(* CODESYS project CtaAppSensor_1.0.0.4.library
   Description: Sensor Library der CTA
   Version: 1.0.0.4
   Title: CtaAppSensor
   Author: SIS
   LanguageModelAttribute: qualified-access-only
   DocFormat: reStructuredText
   Placeholder: CtaAppSensor
   CompiledLibraryCompatibilityVersion: CODESYS V3.5 SP16 Patch 3
   Company: CTA
   DefaultNamespace: CtaAppSensor

Project tree, tasks and I/O mapping:
  libraries: Standard, 3.5.18.0 (System); CtaAppBmk, 1.0.0.0 (CTA); CtaAppReport, 1.0.0.2 (CTA); CtaSysConfig, 1.0.0.2 (CTA); CtaAppFilter, 1.0.0.0 (CTA); VisuSymbols, 4.5.0.0 (System); VisuDialogs, * (System); CtaSysSensorReCalculation, 1.0.0.0 (CTA); CtaVisSymbols, 1.0.0.0 (CTA); CtaAppInfluxLog, 1.0.0.1 (CTA); CtaSysIO, 1.0.0.1 (CTA); CtaVisHelp, 1.0.0.0 (CTA); CtaAppLeistungventile, 1.0.0.0 (CTA); CtaAppModbusSpezifikation, 1.0.0.0 (CTA)
  40 Visualizations/
    COLLECTOR/
      visualisation VIS_SENSOR_COLLECTOR
      visualisation VIS_SENSOR_COLLECTOR_TEMP
      Help Funktionen/
        visualisation SelSort
        visualisation SortPfeil
    ICON/
      SENSOR_FLAT/
        SENSOR_FLAT_TXT_RIGHT/
          ABOVE/
            visualisation VIS_SENSOR_FLAT_RigthAboveCheckIsEnabled
            visualisation VIS_SENSOR_FLAT_RIGHT_ABOVE
            visualisation VIS_SENSOR_FLAT_RigthAboveCheckQuerry
          BELOW/
            visualisation VIS_SENSOR_FLAT_RIGHT_BELOW
            visualisation VIS_SENSOR_FLAT_RigthBelowCheckIsEnabled
            visualisation VIS_SENSOR_FLAT_RigthBelowCheckQuerry
          MIDDLE/
            visualisation VIS_SENSOR_FLAT_RIGHT_MIDDLE
            visualisation VIS_SENSOR_FLAT_RigthMiddleCheckIsEnabled
            visualisation VIS_SENSOR_FLAT_RigthMiddleCheckQuerry
        SENSOR_FLAT_TXT_LEFT/
          BELOW/
            visualisation VIS_SENSOR_FLAT_LEFT_BELOW
            visualisation VIS_SENSOR_FLAT_LeftBelowCheckIsEnabled
            visualisation VIS_SENSOR_FLAT_LeftBelowCheckQuerry
          ABOVE/
            visualisation VIS_SENSOR_FLAT_LeftAboveCheckQuerry
            visualisation VIS_SENSOR_FLAT_LEFT_ABOVE
            visualisation VIS_SENSOR_FLAT_LeftAboveCheckIsEnabled
          MIDDLE/
            visualisation VIS_SENSOR_FLAT_LeftMiddleCheckIsEnabled
            visualisation VIS_SENSOR_FLAT_LeftMiddleCheckQuerry
            visualisation VIS_SENSOR_FLAT_LEFT_MIDDLE
      SENSOR_BASE/
        ICON/
          Round/
            visualisation SensorRound
          Flat/
            visualisation SensorFlat
          Value/
            visualisation ValueDwnUp
            visualisation ValueUpDwn
      SENSOR_ROUND/
        SENSOR_ROUND_TXT_RIGHT/
          ABOVE/
            visualisation VIS_SENSOR_ROUND_RIGHT_ABOVE
            visualisation VIS_SENSOR_ROUND_RightAboveCheckIsEnabled
            visualisation VIS_SENSOR_ROUND_RightAboveCheckQuerry
          BELOW/
            visualisation VIS_SENSOR_ROUND_RIGHT_BELOW
            visualisation VIS_SENSOR_ROUND_RightBelowCheckQuerry
            visualisation VIS_SENSOR_ROUND_RightBelowCheckIsEnabled
        SENSOR_ROUNF_TXT_LEFT/
          ABOVE/
            visualisation VIS_SENSOR_ROUND_LEFT_ABOVE
            visualisation VIS_SENSOR_ROUND_LeftAboveCheckIsEnabled
            visualisation VIS_SENSOR_ROUND_LeftAboveCheckQuerry
          BELOW/
            visualisation VIS_SENSOR_ROUND_LEFT_BELOW
            visualisation VIS_SENSOR_ROUND_LeftBelowCheckIsEnabled
            visualisation VIS_SENSOR_ROUND_LeftBelowCheckQuerry
    POPUP/
      visualisation POPUP_SENSOR
      PARAMETER/
        visualisation VIS_SENSOR_PARAMETER
        visualisation VIS_SENSOR_PARAMETER_LISTE
        SENSOR_ParameterBase/
          visualisation VIS_SENSOR_PARAMETER_BASE0
          visualisation VIS_SENSOR_PARAMETER_BASE
        SENSOR_ReportManagement/
          visualisation Sensor_LowAlarm_Param
          visualisation Sensor_HighAlarm_Param
          visualisation Sensor_HighWarning_Param
          visualisation VIS_SENSOR_PARAMETER_REPORTMNG
          visualisation VIS_SENSOR_PARAMETER_REPORTMNG_1
          visualisation Sensor_LowWarning_Param
        SENSOR_InfluxDb/
          visualisation VIS_SENSOR_PARAMETER_TRENDLOG
          visualisation VIS_SENSOR_PARAMETER_TRENDLOG0
        SENSOR_Filter/
          visualisation VIS_SENSOR_PARAMETER_FILTER
          visualisation VIS_SENSOR_PARAMETER_FILTER_1
        IO_Parameter/
          visualisation VIS_SENSOR_IO_PARAMETER
      visualisation VIS_SENSOR_LISTE
      MANUAL/
        visualisation VIS_SENSOR_MANUAL
      OVERVIEW/
        visualisation VIS_SENSOR_OVERVIEW
        visualisation VIS_SENSOR_OVERVIEW0
      REPORTS/
        visualisation VIS_SENSOR_REPORTS
      BUS/
        visualisation Sensor_BUS_CS
        visualisation Sensor_BUS
        visualisation Sensor_BUS_SW0_Detail
        visualisation Sensor_BUS_SW1_Detail
        visualisation Sensor_BUS_SW2_Detail
        visualisation Sensor_BUS_SW3_Detail
  30 Program Organization Units/
    Abstracte Bausteine/
      function block fbSensorTabellenInfo [ST]: proStateSymbol, proSoftwareValue, proRawValue, proEnSymbol, proPhysicalValue
    fb's/
      Sensor/
        function block fbSensor [ST]: proModulType, actReport, proITF_REPORTMANAGER, actErrorCondition, proLockDown, proAvailable, proAcknowlege, proAtIconNr, actTrendLog, proEn, proEnSymbol, metSetReal, metSetBool, proIsEnabled, proIsError, proStateSymbol, proCountedError, proCountedInfo, proCountedWarning, actState, proInvertierung, proxErrorConditionValue, proConfigError, actConfig, P_scAnalogAlarm_fbxEnableOverflowAl, P_scAnalogAlarm_fbxEnableUnderflowAl, P_scBase_fbxEnable, P_scVisu_fbusiDezimalPos, P_scAlCondition_fbxEnable, P_scAlCondition_fbtDelayTillCondition, P_scHighAlarm_fbiRetryTillLock, P_scHighAlarm_fbiTypeOfAcknolage, P_scHighAlarm_fbrHysterese, P_scHighAlarm_fbrValue, P_scHighAlarm_fbtDelayTillAlarm, P_scHighAlram_fbxDoesAlarm, P_scHighWarning_fbrValue, P_scHighWarning_fbtDelayTillWarning, P_scHighWarning_fbxDoesWarning, P_scInfluxDb_fbxEnable, P_scLoAlarm_fbiRetryTillLock, P_scLoAlarm_fbiTypeOfAcknolage, P_scLoAlarm_fbrHysterese, P_scLoAlarm_fbrValue, P_scLoAlarm_fbtDelayTillAlarm, P_scLoAlarm_fbxDoesAlarm, P_scLoWarning_fbrValue, P_scLoWarning_fbtDelayTillWarning, P_scLoWarning_fbxDoesWarning, P_scManual_fbrManualOnY, P_scManual_fbuiManualControl, P_scManual_fbuiManualState, P_scManual_fbxAllowManualOn, P_scAlarmReset_fbtDealyTillReset, P_scFilter_fbrValue, P_scFilter_fbxEnabled, proSensorITF, proRawValue, FB_INIT, proSoftwareValue, proIsWarning, proIsHandOnOrOff, proIsReady, proHandOff, proHandOn, proHandOnY, proAuto, proManualTrue, proManualFalse, proValueInputType, metSetITF, actDigital, actAnalog, proPhysicalValue, actReCalculate, ITF_RC, actMbState, proModbusTest, proModbusStateWord, proModbusControllWord, prorValue
      Collector/
        function block fbSensor_Collector [ST]: metRegistry, proMin, proMax, proaySensorTabelle, proMissedBuffer, proBufferError, proayAntrieb, metSortArray, metGetAntriebITF
    fc's/
      function fcGetBigerStringValue [ST]
      AlarmControll/
        function fcHighControl [ST]
        function fcLowControl [ST]
      Visu/
        function fcCheckQuerryAndIconReturn [ST]
  00000000-0000-0000-0000-000000000000|D:\CoDeSys\LibrariesV3\trunk\Intern\CAA\CAA Template\3.4.0.0 draft\Placeholder.xml
  00000000-0000-0000-0000-000000000000|D:\CoDeSys\LibrariesV3\trunk\Intern\CAA\CAA Template\3.2.0.3 draft\Prefix.pdf
  00000000-0000-0000-0000-000000000000|D:\CoDeSys\LibrariesV3\trunk\Intern\CAA\CAA Template\3.5.2.0 draft\Placeholder.xml
  20 Structs/
    13 Globale Variablen/
      global variables GVL_SENSOR
    data type scParameter
    LowWarning/
      data type scLoWarning
    BASE/
      data type scBase
    Alarme/
      data type scAnalogAlarm
      Zusatzbedingungen/
        data type scAlCondition
      AlarmReset/
        data type scAlarmReset
    HighWarning/
      data type scHighWarning
    InfluxDb/
      data type scInfluxDb
    Filter/
      data type scFilter
    HighAlarm/
      data type scHighAlarm
    LowAlarm/
      data type scLoAlarm
    Manual/
      data type scManual
    data type enInputType
    Visu/
      data type scVisu
  50 Images/
  10 Documenation/
    global variables VersionHistory
    global variables readMe
  21 Interface/
    interface ITF_SENSOR_COLLECTOR: proBufferError, metGetAntriebITF, proMissedBuffer, proMin, proMax, proaySensorTabelle, metSortArray
    interface ITF_SENSOR_TABELLE_INFO: proRawValue, proSoftwareValue, proEnSymbol, proStateSymbol, proPhysicalValue
    interface ITF_SENSOR: proConfigError, P_scBase_fbxEnable, P_scVisu_fbusiDezimalPos, P_scManual_fbxAllowManualOn, P_scManual_fbuiManualState, P_scManual_fbuiManualControl, P_scManual_fbrManualOnY, P_scFilter_fbxEnabled, P_scFilter_fbrValue, P_scLoWarning_fbxDoesWarning, P_scLoWarning_fbrValue, P_scLoWarning_fbtDelayTillWarning, P_scLoAlarm_fbxDoesAlarm, P_scLoAlarm_fbrValue, P_scLoAlarm_fbrHysterese, P_scLoAlarm_fbtDelayTillAlarm, P_scLoAlarm_fbiRetryTillLock, P_scLoAlarm_fbiTypeOfAcknolage, P_scHighWarning_fbxDoesWarning, P_scHighWarning_fbrValue, P_scHighWarning_fbtDelayTillWarning, P_scHighAlram_fbxDoesAlarm, P_scHighAlarm_fbrValue, P_scHighAlarm_fbrHysterese, P_scHighAlarm_fbtDelayTillAlarm, P_scHighAlarm_fbiRetryTillLock, P_scHighAlarm_fbiTypeOfAcknolage, P_scInfluxDb_fbxEnable, P_scAnalogAlarm_fbxEnableOverflowAl, P_scAnalogAlarm_fbxEnableUnderflowAl, P_scAlCondition_fbxEnable, P_scAlCondition_fbtDelayTillCondition, P_scAlarmReset_fbtDealyTillReset, proSensorITF, proCountedError, proCountedInfo, proITF_REPORTMANAGER, proCountedWarning, proIsHandOnOrOff, proHandOn, proIsError, proIsWarning, proEn, proIsEnabled, proHandOff, proHandOnY, proIsReady, proAuto, proManualFalse, proManualTrue, proValueInputType, proxErrorConditionValue, proInvertierung, prorValue, proLockDown, proAvailable, proAcknowlege, proAtIconNr, ITF_RC, proModbusStateWord, proModbusTest, proModbusControllWord
  11 Library Parameter/
    global variables Parameter
  12 Konstanten/
    global variables GlobalKonstant
  60 Textlisten/
    text list Info
    Types/
      text list WarnungsStatus
      text list ValueInputType
    Reports/
      text list Error
      text list Warnung
  text list GlobalTextList
  5ce3da45-db07-42e7-a21c-a00fff4ed8f6|C:\Users\sis\Downloads\dip-switch.svg
  5ce3da45-db07-42e7-a21c-a00fff4ed8f6|C:\Users\sis\Downloads\lightning-bolt-circle.svg
  5ce3da45-db07-42e7-a21c-a00fff4ed8f6|C:\Users\sis\Downloads\sine-wave.svg
  5ce3da45-db07-42e7-a21c-a00fff4ed8f6|C:\Users\sis\Downloads\eye.svg
  5ce3da45-db07-42e7-a21c-a00fff4ed8f6|C:\Users\sis\Downloads\lan.svg
*)

// 20 Structs/scParameter
{attribute 'pack_mode' := '1'} 
TYPE scParameter :
    STRUCT
        scBase              :   scBase;
		scManual			:	scManual;
		scFilter			:	scFilter;
		scLoWarning			:	scLoWarning;
		scLoAlarm			:	scLoAlarm;
		scHighWarning		:	scHighWarning;
		scHighAlarm			:	scHighAlarm;
		scInfluxDb			:	scInfluxDb;
		scAnalogAlarm		:	scAnalogAlarm;
		scAlCondition		:	scAlCondition;
		scAlarmReset		:	scAlarmReset;
		scVisu				:	scVisu;
    END_STRUCT
END_TYPE

// 20 Structs/HighWarning/scHighWarning
TYPE scHighWarning :
	STRUCT
		fbxDoesWarning			:	CtaSysConfig.fbBOOL;
		fbrValue				:	CtaSysConfig.fbREAL;
		fbtDelayTillWarning		:	CtaSysConfig.fbTIME;	
	END_STRUCT
END_TYPE

// 20 Structs/HighAlarm/scHighAlarm
TYPE scHighAlarm :
	STRUCT
		fbxDoesAlarm			:	CtaSysConfig.fbBOOL;
		fbrValue				:	CtaSysConfig.fbREAL;
		fbrHysterese			:	CtaSysConfig.fbREAL;
		fbtDeleayTillAlarm		:	CtaSysConfig.fbTIME;
		fbiRetryTillLock		:	CtaSysConfig.fbINT;
		fbiTypeOfAcknolage		:	CtaSysConfig.fbINT;
	END_STRUCT
END_TYPE

// 20 Structs/LowAlarm/scLoAlarm
TYPE scLoAlarm :
	STRUCT
		fbxDoesAlarm			:	CtaSysConfig.fbBOOL;
		fbrValue				:	CtaSysConfig.fbREAL;
		fbrHysterese			:	CtaSysConfig.fbREAL;
		fbtDeleayTillAlarm		:	CtaSysConfig.fbTIME;
		fbiRetryTillLock		:	CtaSysConfig.fbINT;
		fbiTypeOfAcknolage		:	CtaSysConfig.fbINT;
	END_STRUCT
END_TYPE

// 20 Structs/LowWarning/scLoWarning
TYPE scLoWarning :
	STRUCT
		fbxDoesWarning			:	CtaSysConfig.fbBOOL;
		fbrValue				:	CtaSysConfig.fbREAL;
		fbtDelayTillWarning		:	CtaSysConfig.fbTIME;		
	END_STRUCT
END_TYPE

// 20 Structs/Alarme/scAnalogAlarm
TYPE scAnalogAlarm :
	STRUCT
		fbxEnableOverflowAl		:	CtaSysConfig.fbBOOL;
		fbxEnableUnderflowAl	:	CtaSysConfig.fbBOOL;
	END_STRUCT
END_TYPE

// 20 Structs/Filter/scFilter
TYPE scFilter :
	STRUCT
		fbxEnabled	:	CtaSysConfig.fbBOOL;
		fbrValue	:	CtaSysConfig.fbREAL;
	END_STRUCT
END_TYPE

// 20 Structs/BASE/scBase
{attribute 'pack_mode' := '1'} 
TYPE scBase :
    STRUCT
        fbxEnable       :   CtaSysConfig.fbBOOL;
    END_STRUCT
END_TYPE

// 20 Structs/InfluxDb/scInfluxDb
{attribute 'pack_mode' := '1'} 
TYPE scInfluxDb :
    STRUCT
        fbxEnable       :   CtaSysConfig.fbBOOL;
    END_STRUCT
END_TYPE

// 20 Structs/Alarme/Zusatzbedingungen/scAlCondition
TYPE scAlCondition :
	STRUCT
		fbxEnable				:	CtaSysConfig.fbBOOL;
		fbtDelayTillCondition	:	CtaSysConfig.fbTIME;
	END_STRUCT
END_TYPE

// 20 Structs/Alarme/AlarmReset/scAlarmReset
TYPE scAlarmReset :
	STRUCT
		fbtDelayTillReset	:	CtaSysConfig.fbTIME;		
	END_STRUCT
END_TYPE

// 20 Structs/Manual/scManual
TYPE scManual :
	STRUCT
		fbxAlowManualOn		:	CtaSysConfig.fbBOOL;
		fbuiManualState		:	CtaSysConfig.fbUINT;
		fbuiManualControl	:	CtaSysConfig.fbUINT;
		fbrManualOnY		:	CtaSysConfig.fbREAL;
	END_STRUCT
END_TYPE

// 20 Structs/enInputType
{attribute 'qualified_only'}
{attribute 'strict'}
TYPE enInputType :
(
	Default := 0,
	AnalogInput,
	DigitalInput,
	Analog_ITF_Input,
	Digital_ITF_Input	
);
END_TYPE

// 20 Structs/Visu/scVisu
TYPE scVisu :
	STRUCT
		fbusiDezimalPos		:	CtaSysConfig.fbUSINT;
	END_STRUCT
END_TYPE

// 10 Documenation/VersionHistory
(* 

.. image:: ../../Images/CTA_Logo.jpg
   :align: right
   :width: 15% 

**Vorlage**   


============ =========== =========== ============================================
**Date**     **Version** **Author**  **Change**
------------ ----------- ----------- --------------------------------------------
04.03.2021   0.0.0.0     SIS         Vorlage erstellt

============ =========== =========== ============================================


*)
VAR_GLOBAL
    stInfo : STRING:= '0.0.0.0, Vorlage, CTA';
END_VAR

// 10 Documenation/readMe
(*

**ReadMe**
 
|	**Empfehlung**
|
|	Bibliothek CtaAppSensor zur auswertung von Sensoren
|	Instanzieren Sie den CtaAppSensor.fbSensor in ihrem Funktionsbaustein oder POU beispielsweise als fbTFühlX (X = Nr.) 
|	Deklarieren Sie die Struktur Variable welche als Parameter und zur ansteuerung dienen wie im Code beispiel.
|  
| *Beispiel* 

+-----------------------+---------------------------------------------------------------------------------------------------------------------------------------------------------------------------------------------------------------------------------------------------------------------------------------------------------------------------------------------------------------------------------------------------------------------------------------+
| Beschreibung          |  Code                                                                                                                                                                                                                                                                                                                                                                                                                                 |
+=======================+=======================================================================================================================================================================================================================================================================================================================================================================================================================================+
| POU oder SmFb         | .. code-block:: codesys                                                                                                                                                                                                                                                                                                                                                                                                               |
|                       |                                                                                                                                                                                                                                                                                                                                                                                                                                       |
|                       |	// Deklaration als VAR im POU oder dem selbsterstellten Funktionsbaustein                                                                                                                                                                                                                                                                                                                                                        	|
|                       |   VAR   																																																				 																																																				|
|						|	    (*Temperaturfühler 1*)																																																		 																																																	|
|						|		fbTFühl1			: CtaAppSensor.fbSensor;                                                                                                                                                                                                                                                                                                                                                               						|
|			 			|	END_VAR                                                                                                                                                                                                                                                                                                                                                                                                                          	|
+-----------------------+---------------------------------------------------------------------------------------------------------------------------------------------------------------------------------------------------------------------------------------------------------------------------------------------------------------------------------------------------------------------------------------------------------------------------------------+
| Code für Init         | .. code-block:: codesys                                                                                                                                                                                                                                                                                                                                                                                                               |
|                       |   																																																					 																																																				|
|			 			|	// Kopieren des nachfolgenden Codes in eine Action zur Initialisierung der Parameter. Zum Beispiel actConfig.																																																				 																										|
|                       |	{region "Parameter Temperaturfühler 1"}                                                                                                                                                                                                                                                                                                                                                                                             |
|			 			|		(*Basis*)                                                                                                                                                                                                                                                                                                                                                                                                                       |
|						|		fbTFühl1.scParameter.scBase.fbxEnable                			(_WertInit :=  TRUE																		 );		//P1 Ein- Ausschalten des Sensors                                                                                                                                                                                                                               |
|						|		(*Handansteuerung*)                                                                                                                                                                                                                                                                                                                                                                                                             |
|						|		fbTFühl1.scParameter.scManual.fbxAlowManualOn					(_WertInit := FALSE																		 );     //P2 Handansteuerung zulassen / nicht zulassen                                                                                                                                                                                                                  |
|						|		fbTFühl1.scParameter.scManual.fbuiManualState					(_WertInit :=	  0									, _MinInit :=     0, _MaxInit:=     2);     //P3 Ansteuerungsmodus des Sensors (auto, manuell, gesperrt)                                                                                                                                                                                                    |
|						|		fbTFühl1.scParameter.scManual.fbuiManualControl					(_WertInit :=     0									, _MinInit :=     0, _MaxInit:=     1);     //P4 Ansteuerungsignal des Sensors (TRUE,FALSE)                                                                                                                                                                                                                 |
|						|		fbTFühl1.scParameter.scManual.fbrManualOnY						(_WertInit :=   0.0									, _MinInit :=      , _MaxInit:=      );     //P5 Manueller Stellwert für den SEnsor                                                                                                                                                                                                                         |
|						|		(*Filter*)                                                                                                                                                                                                                                                                                                                                                                                                                      |
|						|		fbTFühl1.scParameter.scFilter.fbxEnabled						(_WertInit := FALSE																		 );		//P6 Ein- Ausschalten des Filters                                                                                                                                                                                                                               |
|						|		fbTFühl1.scParameter.scFilter.fbrValue							(_WertInit :=   0.0									, _MinInit :=      , _MaxInit:=      );		//P7 Filterwert                                                                                                                                                                                                                                                 |
|						|		(*LowWarning*)                                                                                                                                                                                                                                                                                                                                                                                                                  |
|						|		fbTFühl1.scParameter.scLoWarning.fbxDoesWarning					(_WertInit := FALSE																		 );		//P8 Ein- Ausschalten der LowWarning                                                                                                                                                                                                                            |
|						|		fbTFühl1.scParameter.scLoWarning.fbrValue						(_WertInit :=   0.0									, _minInit :=      , _maxInit:= 	 );		//P9 Wert bei welcher die LowWarning ausgelöst wird                                                                                                                                                                                                             |
|						|		fbTFühl1.scParameter.scLoWarning.fbtDelayTillWarning			(_WertInit :=  T#0S									, _minInit :=      , _maxInit:=      );		//P10 Verzögerungszeit für die Ausgabe des LowWarining Fehlers                                                                                                                                                                                                  |
|						|		(*LowAlarm*)                                                                                                                                                                                                                                                                                                                                                                                                                    |
|						|		fbTFühl1.scParameter.scLoAlarm.fbxDoesAlarm						(_WertInit := FALSE																		 );		//P11 Ein- Ausschalten des LowAlarm                                                                                                                                                                                                                             |
|						|		fbTFühl1.scParameter.scLoAlarm.fbrValue							(_WertInit :=   0.0									, _minInit :=      , _maxInit:= 	 );		//P12 Wert bei welchem der LowAlarm ausgelöst wird                                                                                                                                                                                                              |
|						|		fbTFühl1.scParameter.scLoAlarm.fbrHysterese						(_WertInit :=   0.0									, _minInit :=      , _maxInit:= 	 );		//P13 Histerese welche zur Rücksetung des Fehlers erreicht werden muss                                                                                                                                                                                          |
|						|		fbTFühl1.scParameter.scLoAlarm.fbtDeleayTillAlarm				(_WertInit :=  T#0S									, _minInit :=      , _maxInit:= 	 );		//P14 Verzögerungszeit für die Ausgabe des LowAlarm Fehlers                                                                                                                                                                                                     |
|						|		fbTFühl1.scParameter.scLoAlarm.fbiTypeOfAcknolage				(_WertInit :=     0 								, _minInit :=     0, _maxInit:=     2);		//P15 Art der Quittierung des Fehlers (auto, quittierned, quittiernd bis n Meldung)                                                                                                                                                                             |
|						|		fbTFühl1.scParameter.scLoAlarm.fbiRetryTillLock					(_WertInit :=     3									, _minInit :=     0, _maxInit:=     5);		//P16 Maximale Anzahl Wiederholungen bis zu Sperrung der Anlage                                                                                                                                                                                                 |
|						|		(*HighWarning*)                                                                                                                                                                                                                                                                                                                                                                                                                 |
|						|		fbTFühl1.scParameter.scHighWarning.fbxDoesWarning				(_WertInit := FALSE																		 );		//P17 Ein- Ausschalten der HighWarning                                                                                                                                                                                                                    		|
|						|		fbTFühl1.scParameter.scHighWarning.fbrValue						(_WertInit :=   0.0									, _minInit :=      , _maxInit:= 	 );		//P18 Wert bei welcher die HighWarning ausgelöst wird                                                                                                                                                                                                     		|
|						|		fbTFühl1.scParameter.scHighWarning.fbtDelayTillWarning			(_WertInit :=  T#0S									, _minInit := 	   , _maxInit:= 	 );		//P19 Verzögerungszeit für die Ausgabe des HighWarining Fehlers                                                                                                                                                                                           		|
|						|		(*HighAlarm*)                                                                                                                                                                                                                                                                                                                                                                                                                   |
|						|		fbTFühl1.scParameter.scHighAlarm.fbxDoesAlarm					(_WertInit := FALSE															 			 );		//P20 Ein- Ausschalten des HighAlarm                                                                                                                                                                                                                            |
|						|		fbTFühl1.scParameter.scHighAlarm.fbrValue						(_WertInit :=   0.0									, _minInit :=      , _maxInit:=      );		//P21 Wert bei welchem der HighAlarm ausgelöst wird                                                                                                                                                                                                             |
|						|		fbTFühl1.scParameter.scHighAlarm.fbrHysterese					(_WertInit :=   0.0									, _minInit :=      , _maxInit:= 	 );		//P22 Histerese welche zur Rücksetung des Fehlers erreicht werden muss                                                                                                                                                                                          |
|						|		fbTFühl1.scParameter.scHighAlarm.fbtDeleayTillAlarm				(_WertInit :=  T#0S									, _minInit :=      , _maxInit:=      );		//P23 Verzögerungszeit für die Ausgabe des HighAlarm Fehlers                                                                                                                                                                                                    |
|						|		fbTFühl1.scParameter.scHighAlarm.fbiTypeOfAcknolage				(_WertInit := 	  0 								, _minInit :=      , _maxInit:=     2);		//P24 Art der Quittierung des Fehlers (auto, quittierned, quittiernd bis n Meldung)                                                                                                                                                                             |
|						|		fbTFühl1.scParameter.scHighAlarm.fbiRetryTillLock				(_WertInit :=     3									, _minInit :=      , _maxInit:=     5);		//P25 Maximale Anzahl Wiederholungen bis zu Sperrung der Anlage                                                                                                                                                                                                 |
|						|		(*Überlauf, Unterlauf*)                                                                                                                                                                                                                                                                                                                                                                                                         |
|						|		fbTFühl1.scParameter.scAnalogAlarm.fbxEnableOverflowAl			(_WertInit :=  TRUE																		 );		//P26 Ein- Ausschalten des Überlauf- Alarms                                                                                                                                                                                                                     |
|						|		fbTFühl1.scParameter.scAnalogAlarm.fbxEnableUnderflowAl			(_WertInit :=  TRUE																		 );		//P27 Ein- Ausschalten des Unterlauf- Alrams                                                                                                                                                                                                                    |
|						|		(*Zusatzbedingung*)                                                                                                                                                                                                                                                                                                                                                                                                             |
|						|		fbTFühl1.scParameter.scAlCondition.fbxEnable 					(_WertInit := FALSE																		 );		//P28 Ein- Ausschalten der Zusatzbedingung                                                                                                                                                                                                                      |
|						|		fbTFühl1.scParameter.scAlCondition.fbtDelayTillCondition		(_WertInit :=  T#0S									, _minInit :=      ,_maxInit:=       );		//P29 Verzögerung für die Zusatzbedingung                                                                                                                                                                                                                       |
|						|		(*Alarmrücksetzung*)                                                                                                                                                                                                                                                                                                                                                                                                            |
|						|		fbTFühl1.scParameter.scAlarmReset.fbtDelayTillReset				(_WertInit := T#24H									, _minInit :=      ,_maxInit:=       );		//P30 Verzögerung für die Fehlerrücksetzung                                                                                                                                                                                                                     |
|						|		(*Trendlog*)                                                                                                                                                                                                                                                                                                                                                                                                                    |
|						|		fbTFühl1.scParameter.scInfluxDb.fbxEnable            			(_WertInit := TRUE																		 );		//P31 Aktiverung / Deaktivierung der Trenddaten														 																																							|
|						|		(*Visu*)                                                                                                                                                                                                                                                                                                                                                                                                                    	|
|						|		fbTFühl1.scParameter.scVisu.fbusiDezimalPos            			(_WertInit :=     1									, _minInit := 0     , _maxInit:=    3);		//P32 Dezimalstellen auf Visu													 																																												|
|						|	{endregion}                                                                                                                                                      																																																																    | 
|						|																																																																																																										|
+-----------------------+---------------------------------------------------------------------------------------------------------------------------------------------------------------------------------------------------------------------------------------------------------------------------------------------------------------------------------------------------------------------------------------------------------------------------------------+
*)                                                                                                                                                                                                                                                                                                                                                                                                                                                               
VAR_GLOBAL
	xReadMeDone              :   BOOL; 
END_VAR

// 20 Structs/13 Globale Variablen/GVL_SENSOR
{attribute 'qualified_only'}
VAR_GLOBAL
    fbSENSOR_COLLECTOR	:   fbSensor_Collector;   
    xValidData          :   BOOL;
END_VAR

// 11 Library Parameter/Parameter
{attribute 'qualified_only'}
VAR_GLOBAL CONSTANT
    iMaxSensor :   INT   := 60;         // Maximale Anzahl verwendeter AT-Bausteine    
END_VAR

// 12 Konstanten/GlobalKonstant
{attribute 'qualified_only'}
VAR_GLOBAL CONSTANT 	
	stReportTextListError   : CtaAppReport.stReportTextList := 'CtaAppSensor.Error';
	stReportTextListWarning : CtaAppReport.stReportTextList := 'CtaAppSensor.Warnung';
	stReportTextListInfo    : CtaAppReport.stReportTextList := 'CtaAppSensor.Info';	
END_VAR

// 30 Program Organization Units/fb's/Sensor/fbSensor
FUNCTION_BLOCK fbSensor EXTENDS fbSensorTabellenInfo IMPLEMENTS ITF_SENSOR 
VAR_INPUT
    xAlCondition               	:   BOOL;
	xEnHandMode					:	BOOL;
 	rSimValue					:	REAL;
END_VAR                         
VAR_OUTPUT 
    xValue                      :   BOOL;
    rValue						:   REAL;
	rValueRC					:	REAL;
	xIsHandMode					:	BOOL;
END_VAR                 
VAR 
	(*Inputs*)
	ITF_IO_IN					:	CtaSysIO.ITF_IO;
	xValueIn					:	BOOL;
	rValueIn					:	REAL;	
	(* Input Type*)
	xIsITF						:	BOOL;
	xIsBool						:	BOOL;
	xIsReal						:	BOOL;
    stAlternateUnit				:	STRING(5);                
    (* State Intern*)
	xIsDigital					:	BOOL;
	_ITF_DI						: 	CtaSysIO.ITF_DI;
	_ITF_AI						:	CtaSysIO.ITF_AI; 	
	rValueTemp					:	REAL;
	xValueTemp					:	BOOL;
	enValueInputType			:   enInputType;     
    scEWI                       :   CtaAppReport.scReportNr; 
	xIsEnabled					:	BOOL;                
	xConfigError                :   BOOL;
	uiIconNr					:	UINT;
	xOk							:	BOOL;
	(* Modbus *)
    xModbusTest                 :   BOOL;
    ayMbControllWord            :   ARRAY[0..3] OF WORD;
    ayMbStateWord               :   ARRAY[0..3] OF WORD;	
    (* Parameter *)
    fbConfigFile                :   CtaSysConfig.fbConfigFile;
    scParameter                 :   scParameter;	
    (* Reports *)		
    fbReportManager			    :   CtaAppReport.fbReportManager;      
    difor					    :	DINT;                                                                    
    ayErrorReporter				:	ARRAY[1..7] OF CtaAppReport.fbReporter;
	ayWarningReporter			:	ARRAY[1..6] OF CtaAppReport.fbReporter; 	
	_xIsWarning					:	BOOL;
	xIsWarning					:	BOOL;	
	_xIsError					:	BOOL;
	xIsError					:	BOOL;		
	xLoWarning					:	BOOL;
	xLoAlarm					:	BOOL;
	xHiWarning					:	BOOL;
	xHiAlarm					:	BOOL;	
	(* Trendlogs *)
	fbTrendxValue				:	CtaAppInfluxLog.FB_LOG_NODE_BOOL;
	fbTrendrValue				:	CtaAppInfluxLog.FB_LOG_NODE_REAL;
	fbTrendrVaueUnfiltered		:	CtaAppInfluxLog.FB_LOG_NODE_REAL;
	fbTrendrVaueRC				:	CtaAppInfluxLog.FB_LOG_NODE_REAL;
	(* Filter *)
	fbFilter					:	CtaAppFilter.fbImpulsFilter;	
	rValueUngefiltert			:	REAL;	
    (* Collector *)
    diArrayPosition             :   DINT;
	xManualValue				:	BOOL;
	xIsHandOff					:	BOOL;
	xIsHandOn					:	BOOL;
	xIsAuto						:	BOOL;
	xIsHand						:	BOOL;
	TON_DelayAlCondition		: 	TON;
	xErrorConditionOn			: 	BOOL;
	
	xErrorConditionAttached		:	BOOL;
	(*Calculator *)				
	ITF_RC_QUERY				:	CtaSysSensorReCalculation.ITF_SENSOR_RE_CALCULATE;
END_VAR

(* Config *)
actConfig();

(* Sensor Command *)
IF xIsEnabled AND NOT xConfigError THEN
	IF xIsITF THEN
		IF __QUERYINTERFACE(ITF_IO_IN,_ITF_DI) THEN
			enValueInputType := enInputType.Digital_ITF_Input;
			actDigital();
		ELSIF __QUERYINTERFACE(ITF_IO_IN,_ITF_AI) THEN
			enValueInputType := enInputType.Analog_ITF_Input;
			actAnalog();
		END_IF
		
	ELSIF xIsBool THEN
		enValueInputType := enInputType.DigitalInput;
		actDigital();
	ELSIF xIsReal THEN
		enValueInputType := enInputType.AnalogInput;
		actAnalog();
	ELSE
		enValueInputType := enInputType.Default;		
	END_IF	
	
	(* Al Condition *)
    actErrorCondition();	
    (* EWI *)
    actReport();    

	(* Recalculation *)
	actReCalculate();             
ELSE
    IF xConfigError THEN
        (* EWI *)
      actReport();         
	END_IF;
END_IF;

(* State *)
actState();
actMbState();
(* InfluxDB *)
actTrendLog();

PROPERTY proModulType : CtaSysIO.enModuleType
GET
proModulType := ITF_IO_IN.proModuleType;
END_GET
END_PROPERTY

ACTION actReport:
(* EWI Manager *)
fbReportManager(	stErrorInitReportTextListIn		:=	ADR(GlobalKonstant.stReportTextListError),
					stWarningInitReportTextListIn	:=	ADR(GlobalKonstant.stReportTextListWarning),
					stInfoInitReportTextListIn		:=	ADR(GlobalKonstant.stReportTextListInfo),
					scReportNr						:=	scEWI);

IF xIsBool OR (xIsITF AND __QUERYINTERFACE (ITF_IO_IN,_ITF_DI))  THEN
	(* Errors *)                        
        (* Alarm Minimalwert erreicht *)
        ayErrorReporter[1].proPrio  := 2;
        ayErrorReporter[1].metReport(     		xSetReportIn					:= xErrorConditionOn AND scParameter.scLoAlarm.fbxDoesAlarm.proValue AND xLoAlarm,
												iReportID						:= 1,
												enReportTypeIn					:= CtaAppReport.enReportType.Error,  
												enReportAcknowledgeTypeIn   	:= scParameter.scLoAlarm.fbiTypeOfAcknolage.proValue,
												tDelay							:= scParameter.scLoAlarm.fbtDeleayTillAlarm.proValue, 
												ITF_BMK_IN						:= THIS^,			              
												pstReportTextListIn				:= ADR(GlobalKonstant.stReportTextListError),
												stOptionalReportText		    := '',   
												iRetryTilReportLock 		    := scParameter.scLoAlarm.fbiRetryTillLock.proValue, 
												xResetCount         		    := FALSE,  
												tReset						    := scParameter.scAlarmReset.fbtDelayTillReset.proValue); 		

        (* Alarm Maximalwert erreicht *)    
        ayErrorReporter[2].proPrio  := 2;
        ayErrorReporter[2].metReport(     		xSetReportIn					:= xErrorConditionOn AND scParameter.scHighAlarm.fbxDoesAlarm.proValue AND xHiAlarm,
												iReportID						:= 2,
												enReportTypeIn					:= CtaAppReport.enReportType.Error,  
												enReportAcknowledgeTypeIn   	:= scParameter.scHighAlarm.fbiTypeOfAcknolage.proValue,
												tDelay							:= scParameter.scHighAlarm.fbtDeleayTillAlarm.proValue, 
												ITF_BMK_IN						:= THIS^,			              
												pstReportTextListIn				:= ADR(GlobalKonstant.stReportTextListError),
												stOptionalReportText		    := '',   
												iRetryTilReportLock 		    := scParameter.scHighAlarm.fbiRetryTillLock.proValue,
												xResetCount         		    := FALSE, 
	                               				tReset						    := scParameter.scAlarmReset.fbtDelayTillReset.proValue); 		

(* Warnungen *)      
        (* Warnung Minimalwert erreicht *)      
        ayWarningReporter[1].proPrio := 2;
        ayWarningReporter[1].metReport(			xSetReportIn					:= xErrorConditionOn AND scParameter.scLoWarning.fbxDoesWarning.proValue AND xLoWarning,
												iReportID						:= 1,
												enReportTypeIn					:= CtaAppReport.enReportType.Warning,  
												enReportAcknowledgeTypeIn   	:= CtaAppReport.enReportAcknowledgeType.Auto,
												tDelay							:= scParameter.scLoWarning.fbtDelayTillWarning.proValue, 
												ITF_BMK_IN						:= THIS^,			              
												pstReportTextListIn				:= ADR(GlobalKonstant.stReportTextListWarning),
												stOptionalReportText		    := '',   
												iRetryTilReportLock 		    := 0, 
												xResetCount         		    := FALSE,  
												tReset						    := T#0S);                       
                                  
        (* Warnung Maxiwalwert erreicht *)
        ayWarningReporter[2].proPrio := 2;
        ayWarningReporter[2].metReport(			xSetReportIn					:= xErrorConditionOn AND scParameter.scHighWarning.fbxDoesWarning.proValue AND xHiWarning,
												iReportID						:= 2,
												enReportTypeIn					:= CtaAppReport.enReportType.Warning,  
												enReportAcknowledgeTypeIn   	:= CtaAppReport.enReportAcknowledgeType.Auto,
												tDelay							:= scParameter.scHighWarning.fbtDelayTillWarning.proValue, 
												ITF_BMK_IN						:= THIS^,			              
												pstReportTextListIn				:= ADR(GlobalKonstant.stReportTextListWarning),
												stOptionalReportText		    := '',   
												iRetryTilReportLock 		    := 0, 
												xResetCount         		    := FALSE,
												tReset						    := T#0S);  
		
ELSIF xIsReal OR (xIsITF AND __QUERYINTERFACE (ITF_IO_IN,_ITF_AI)) THEN
(* Errors *)                        
	(* Alarm Minimalwert erreicht *)
	ayErrorReporter[3].proPrio  := 2;
	ayErrorReporter[3].metReport(     		xSetReportIn					:= xErrorConditionOn AND scParameter.scLoAlarm.fbxDoesAlarm.proValue AND xLoAlarm,
											iReportID						:= 3,
											enReportTypeIn					:= CtaAppReport.enReportType.Error,  
											enReportAcknowledgeTypeIn   	:= scParameter.scLoAlarm.fbiTypeOfAcknolage.proValue,
											tDelay							:= scParameter.scLoAlarm.fbtDeleayTillAlarm.proValue, 
											ITF_BMK_IN						:= THIS^,			              
											pstReportTextListIn				:= ADR(GlobalKonstant.stReportTextListError),
											stOptionalReportText		    := '',   
											iRetryTilReportLock 		    := scParameter.scLoAlarm.fbiRetryTillLock.proValue, 
											xResetCount         		    := FALSE,  
											tReset						    := scParameter.scAlarmReset.fbtDelayTillReset.proValue); 		

	(* Alarm Maximalwert erreicht *)    
	ayErrorReporter[4].proPrio  := 2;
	ayErrorReporter[4].metReport(     		xSetReportIn					:= xErrorConditionOn AND scParameter.scHighAlarm.fbxDoesAlarm.proValue AND xHiAlarm,
											iReportID						:= 4,
											enReportTypeIn					:= CtaAppReport.enReportType.Error,  
											enReportAcknowledgeTypeIn   	:= scParameter.scHighAlarm.fbiTypeOfAcknolage.proValue,
											tDelay							:= scParameter.scHighAlarm.fbtDeleayTillAlarm.proValue, 
											ITF_BMK_IN						:= THIS^,			              
											pstReportTextListIn				:= ADR(GlobalKonstant.stReportTextListError),
											stOptionalReportText		    := '',   
											iRetryTilReportLock 		    := scParameter.scHighAlarm.fbiRetryTillLock.proValue,
											xResetCount         		    := FALSE, 
											tReset						    := scParameter.scAlarmReset.fbtDelayTillReset.proValue); 
		
		(* Additional errors over interface*)
		IF NOT xIsReal THEN									
			(* Alarm Unterlauf *)
			ayErrorReporter[5].proPrio  := 2;
			ayErrorReporter[5].metReport(     		xSetReportIn					:= scParameter.scAnalogAlarm.fbxEnableUnderflowAl.proValue AND _ITF_AI.proAlUnterlauf,
													iReportID						:= 5,
													enReportTypeIn					:= CtaAppReport.enReportType.Error,  
													enReportAcknowledgeTypeIn   	:= CtaAppReport.enReportAcknowledgeType.Auto,
													tDelay							:= T#0S, 
													ITF_BMK_IN						:= THIS^,			              
													pstReportTextListIn				:= ADR(GlobalKonstant.stReportTextListError),
													stOptionalReportText		    := '',   
													iRetryTilReportLock 		    := 0, 
													xResetCount         		    := FALSE,  
													tReset						    := T#0S); 		
		
			(* Alarm Überlauf *)    
			ayErrorReporter[6].proPrio  := 2;
			ayErrorReporter[6].metReport(     		xSetReportIn					:= scParameter.scAnalogAlarm.fbxEnableOverflowAl.proValue AND _ITF_AI.proAlUeberlauf,
													iReportID						:= 6,
													enReportTypeIn					:= CtaAppReport.enReportType.Error,  
													enReportAcknowledgeTypeIn   	:= CtaAppReport.enReportAcknowledgeType.Auto,
													tDelay							:= T#0S, 
													ITF_BMK_IN						:= THIS^,			              
													pstReportTextListIn				:= ADR(GlobalKonstant.stReportTextListError),
													stOptionalReportText		    := '',   
													iRetryTilReportLock 		    := 0,
													xResetCount         		    := FALSE, 
													tReset						    := T#0S);
		END_IF
			
(* Warnungen *)      
	(* Warnung Minimalwert erreicht *)      
	ayWarningReporter[3].proPrio := 2;
	ayWarningReporter[3].metReport(			xSetReportIn					:= xErrorConditionOn AND scParameter.scLoWarning.fbxDoesWarning.proValue AND xLoWarning,
											iReportID						:= 3,
											enReportTypeIn					:= CtaAppReport.enReportType.Warning,  
											enReportAcknowledgeTypeIn   	:= CtaAppReport.enReportAcknowledgeType.Auto,
											tDelay							:= scParameter.scLoWarning.fbtDelayTillWarning.proValue, 
											ITF_BMK_IN						:= THIS^,			              
											pstReportTextListIn				:= ADR(GlobalKonstant.stReportTextListWarning),
											stOptionalReportText		    := '',   
											iRetryTilReportLock 		    := 0, 
											xResetCount         		    := FALSE,  
											tReset						    := T#0S);                       
							  
	(* Warnung Maxiwalwert erreicht *)
	ayWarningReporter[4].proPrio := 2;
	ayWarningReporter[4].metReport(			xSetReportIn					:= xErrorConditionOn AND scParameter.scHighWarning.fbxDoesWarning.proValue AND xHiWarning,
											iReportID						:= 4,
											enReportTypeIn					:= CtaAppReport.enReportType.Warning,  
											enReportAcknowledgeTypeIn   	:= CtaAppReport.enReportAcknowledgeType.Auto,
											tDelay							:= scParameter.scHighWarning.fbtDelayTillWarning.proValue, 
											ITF_BMK_IN						:= THIS^,			              
											pstReportTextListIn				:= ADR(GlobalKonstant.stReportTextListWarning),
											stOptionalReportText		    := '',   
											iRetryTilReportLock 		    := 0, 
											xResetCount         		    := FALSE,
											tReset						    := T#0S);
END_IF

(* Config Error *)    
ayErrorReporter[7].proPrio  := 1;
ayErrorReporter[7].metReport(     		xSetReportIn					:= xConfigError,
										iReportID						:= 7,
										enReportTypeIn					:= CtaAppReport.enReportType.Error,  
										enReportAcknowledgeTypeIn   	:= CtaAppReport.enReportacknowledgeType.Quit,
										tDelay							:= T#1S, 
										ITF_BMK_IN						:= THIS^,			              
										pstReportTextListIn				:= ADR(GlobalKonstant.stReportTextListError),
										stOptionalReportText		    := '',   
										iRetryTilReportLock 		    := 0, 
										xResetCount         		    := FALSE,  
										tReset						    := T#24H);                            

		
(* Warnung Hand Aus *)      
ayWarningReporter[5].proPrio := 3;  
ayWarningReporter[5].proHandLokal :=    xIsHandOff; 
ayWarningReporter[5].metReport(			xSetReportIn					:= xIsHandOff,
										iReportID						:= 5,
										enReportTypeIn					:= CtaAppReport.enReportType.Warning,  
										enReportAcknowledgeTypeIn   	:= CtaAppReport.enReportAcknowledgeType.Auto,
										tDelay							:= T#0S, 
										ITF_BMK_IN						:= THIS^,			              
										pstReportTextListIn				:= ADR(GlobalKonstant.stReportTextListWarning),
										stOptionalReportText		    := '',   
										iRetryTilReportLock 		    := 0, 
										xResetCount         		    := FALSE,  
										tReset						    := T#24H);                                  
                                
(* Warnung Hand Ein *)    
ayWarningReporter[6].proPrio := 3; 
ayWarningReporter[6].proHandLokal :=    xIsHandOn;
ayWarningReporter[6].metReport(			xSetReportIn					:= xIsHandOn OR xIsHandMode,
										iReportID						:= 6,
										enReportTypeIn					:= CtaAppReport.enReportType.Warning,  
										enReportAcknowledgeTypeIn   	:= CtaAppReport.enReportAcknowledgeType.Auto,
										tDelay							:= T#0S, 
										ITF_BMK_IN						:= THIS^,			              
										pstReportTextListIn				:= ADR(GlobalKonstant.stReportTextListWarning),
										stOptionalReportText		    := '',   
										iRetryTilReportLock 		    := 0, 
										xResetCount         		    := FALSE,  
										tReset						    := T#24H);                                           
	
(* Sync Reports *)                                         
FOR difor := LOWER_BOUND(ayErrorReporter,1) TO UPPER_BOUND(ayErrorReporter,1) DO
	fbReportManager.metSyncReporter(ayErrorReporter[difor]);	
END_FOR;
FOR difor := LOWER_BOUND(ayWarningReporter,1) TO UPPER_BOUND(ayWarningReporter,1) DO
	fbReportManager.metSyncReporter(ayWarningReporter[difor]);	
END_FOR;
                                                                          
_xIsError   := scEWI.iError <> 0;
_xIsWarning := scEWI.iWarning <> 0;
END_ACTION

PROPERTY proITF_REPORTMANAGER : CtaAppReport.ITF_REPORTMANAGER
GET
proITF_REPORTMANAGER := fbReportManager;
END_GET
END_PROPERTY

ACTION actErrorCondition:
//  Zeitverzögerung bis die Alarmierung Freigegeben wird


IF scParameter.scAlCondition.fbxEnable.proValue			THEN
	TON_DelayAlCondition(   PT:=    scParameter.scAlCondition.fbtDelayTillCondition.proValue,
							IN:=	xAlCondition,
							Q=>     xErrorConditionOn);  
             
ELSE
xErrorConditionOn		:=TRUE;	
END_IF
END_ACTION

{attribute 'monitoring' := 'variable'}
PROPERTY proLockDown : BOOL
GET
proLockDown := proIsError;
END_GET
END_PROPERTY

{attribute 'monitoring' := 'variable'}
PROPERTY proAvailable : BOOL
GET
proAvailable := proIsReady;
END_GET
END_PROPERTY

{attribute 'monitoring' := 'variable'}
PROPERTY proAcknowlege : BOOL
GET
proAcknowlege := xValue AND NOT proIsError ;
END_GET
END_PROPERTY

PROPERTY proAtIconNr : UINT
SET
uiIconNr := proAtIconNr;
END_SET
GET
proAtIconNr:= uiIconNr;
END_GET
END_PROPERTY

ACTION actTrendLog:
(* Istwert bool *)
fbTrendxValue.ENABLE		:= 	scParameter.scBase.fbxEnable.proValue AND 
								scParameter.scInfluxDb.fbxEnable.proValue;
fbTrendxValue.KEY           :=  CONCAT(stObjID,'_xValue');
fbTrendxValue.SET_VALUE     :=  xValue;

(* Istwert real *)
fbTrendrValue.ENABLE		:=	scParameter.scBase.fbxEnable.proValue AND 
								scParameter.scInfluxDb.fbxEnable.proValue;
fbTrendrValue.KEY           :=  CONCAT(stObjID,'_rValue');
fbTrendrValue.SET_VALUE     :=  rValue;

IF (xIsITF AND  __QUERYINTERFACE (ITF_IO_IN,_ITF_AI)) OR xIsReal THEN
	(* Istwert real ungefiltert*)
	fbTrendrVaueUnfiltered.ENABLE		:=	scParameter.scBase.fbxEnable.proValue AND 
											scParameter.scInfluxDb.fbxEnable.proValue;
	fbTrendrVaueUnfiltered.KEY			:=  CONCAT(stObjID,'_rValueUnfiltered');
	fbTrendrVaueUnfiltered.SET_VALUE	:= 	rValueUngefiltert;
ELSE
	(* Istwert real ungefiltert*)
	fbTrendrVaueUnfiltered.ENABLE		:=	FALSE;
	fbTrendrVaueUnfiltered.KEY			:=  CONCAT(stObjID,'_rValueUnfiltered');
	fbTrendrVaueUnfiltered.SET_VALUE	:= 	rValueUngefiltert;	
END_IF;

IF __QUERYINTERFACE(ITF_RC_QUERY,ITF_RC_QUERY) THEN
	(* Recalculatet Value Enable*)
	fbTrendrVaueRC.ENABLE				:=	scParameter.scBase.fbxEnable.proValue AND 
											scParameter.scInfluxDb.fbxEnable.proValue;
	fbTrendrVaueRC.KEY					:=  CONCAT(stObjID,'_rValueRecalculatet');
	fbTrendrVaueRC.SET_VALUE			:= 	rValueRC;
ELSE
	(* Recalculatet Value Disable*)
	fbTrendrVaueRC.ENABLE				:=	FALSE;
	fbTrendrVaueRC.KEY					:=  CONCAT(stObjID,'_rValueRecalculatet');
	fbTrendrVaueRC.SET_VALUE			:= 	rValueRC;	
END_IF;
END_ACTION

PROPERTY proEn : BOOL
SET
xIsEnabled := proEn;
END_SET
GET
proEn := xIsEnabled;
END_GET
END_PROPERTY

PROPERTY proEnSymbol : STRING
GET
IF xIsEnabled THEN
    proEnSymbol := 'CtaVisSymbols.ImagePool.CheckboxChecked_blue';
ELSE    
    proEnSymbol := 'CtaVisSymbols.ImagePool.CheckboxUnchecked_withe'; 
END_IF;
END_GET
END_PROPERTY

METHOD metSetReal
VAR_INPUT
	rRealIn				:	REAL;
	stAlternateUnitIn	:	STRING(5);
END_VAR
rValueIn 		:= rRealIn;
xIsITF 			:= FALSE;
xIsBool 		:= FALSE;
xIsReal 		:= TRUE;
stAlternateUnit := stAlternateUnitIn;
END_METHOD

METHOD metSetBool
VAR_INPUT
	xBoolIn		:  BOOL;
END_VAR
xValueIn := xBoolIn;
xIsITF	:= FALSE;
xIsBool := TRUE;
xIsReal := FALSE;
END_METHOD

PROPERTY proIsEnabled : BOOL
GET
proIsEnabled := xIsEnabled;
END_GET
END_PROPERTY

PROPERTY proIsError : BOOL
GET
proIsError := xIsError;
END_GET
END_PROPERTY

PROPERTY proStateSymbol : STRING
GET
IF xIsError THEN
    proStateSymbol := 'CtaVisSymbols.ImagePool.CtaError';
ELSE    
    IF xIsWarning THEN
        IF scEWI.iWarning = 5 THEN
            proStateSymbol := 'CtaVisSymbols.ImagePool.front_hand_Yellow_Off';
        ELSIF scEWI.iWarning = 6 THEN
            proStateSymbol := 'CtaVisSymbols.ImagePool.front_hand_Yellow';
        ELSE
            proStateSymbol := 'CtaVisSymbols.ImagePool.CtaWarning';
        END_IF;
     ELSE
         proStateSymbol := '';
	 END_IF
END_IF;
END_GET
END_PROPERTY

PROPERTY proCountedError : INT
GET
proCountedError := fbReportManager.proAnzError;
END_GET
END_PROPERTY

PROPERTY proCountedInfo : INT
GET
proCountedInfo := fbReportManager.proAnzInfo;
END_GET
END_PROPERTY

PROPERTY proCountedWarning : INT
GET
proCountedWarning := fbReportManager.proAnzWarning;
END_GET
END_PROPERTY

ACTION actState:
xIsWarning      := _xIsWarning;         
xIsError        := _xIsError;        
xIsEnabled      := scParameter.scBase.fbxEnable.proValue;         
xIsHandOn       := scParameter.scManual.fbuiManualState.proValue = 2;         
xIsHandOff      := scParameter.scManual.fbuiManualState.proValue = 1;          
xIsAuto         := scParameter.scManual.fbuiManualState.proValue = 0;
xManualValue	:= scParameter.scManual.fbuiManualControl.proValue = 1 AND scParameter.scManual.fbuiManualControl.proValue <> 0;
xIsHand        	:= xIsHandOn OR xEnHandMode OR xIsHandOff;
END_ACTION

PROPERTY proInvertierung : BOOL;
GET
IF __QUERYINTERFACE(_ITF_DI,_ITF_DI) THEN	
	proInvertierung := 	TO_BOOL(CtaSysConfig.fcGetEnumerationId(_ITF_DI.P_scfbDI_fbxInvert));
ELSE
	proInvertierung := FALSE;
END_IF
END_GET
END_PROPERTY

PROPERTY proxErrorConditionValue : BOOL
GET
proxErrorConditionValue := xErrorConditionOn;
END_GET
END_PROPERTY

PROPERTY proConfigError : BOOL
GET
proConfigError := xConfigError;
END_GET
END_PROPERTY

ACTION actConfig:
(* Config Fb *)
fbConfigFile();

(* Base Parameter *)
scParameter.scBase.fbxEnable                			(_usiParaNr :=  1, ItfConfigFb := fbConfigFile);

(* Manual *)
scParameter.scManual.fbxAlowManualOn					(_usiParaNr :=  2, itfConfigFb := fbConfigFile);
scParameter.scManual.fbuiManualState					(_usiParaNr :=  3, itfConfigFb := fbConfigFile);
scParameter.scManual.fbuiManualControl					(_usiParaNr :=  4, itfConfigFb := fbConfigFile);
scParameter.scManual.fbrManualOnY						(_usiParaNr :=  5, itfConfigFb := fbConfigFile);

(* Filter *)
scParameter.scFilter.fbxEnabled							(_usiParaNr :=  6, itfConfigFb := fbConfigFile);
scParameter.scFilter.fbrValue							(_usiParaNr :=  7, itfConfigFb := fbConfigFile);

(* Low warning *)
scParameter.scLoWarning.fbxDoesWarning					(_usiParaNr :=  8, itfConfigFb := fbConfigFile);
scParameter.scLoWarning.fbrValue						(_usiParaNr :=  9, itfConfigFb := fbConfigFile);
scParameter.scLoWarning.fbtDelayTillWarning				(_usiParaNr := 10, itfConfigFb := fbConfigFile);

(* Low alarm *)
scParameter.scLoAlarm.fbxDoesAlarm						(_usiParaNr := 11, itfConfigFb := fbConfigFile);
scParameter.scLoAlarm.fbrValue							(_usiParaNr := 12, itfConfigFb := fbConfigFile);
scParameter.scLoAlarm.fbrHysterese						(_usiParaNr := 13, itfConfigFb := fbConfigFile);
scParameter.scLoAlarm.fbtDeleayTillAlarm				(_usiParaNr := 14, itfConfigFb := fbConfigFile);
scParameter.scLoAlarm.fbiTypeOfAcknolage				(_usiParaNr := 15, itfConfigFb := fbConfigFile, _MinInit := 0 , _MaxInit := 2);
scParameter.scLoAlarm.fbiRetryTillLock					(_usiParaNr := 16, itfConfigFb := fbConfigFile);

(* High warning *)
scParameter.scHighWarning.fbxDoesWarning				(_usiParaNr := 17, itfConfigFb := fbConfigFile);
scParameter.scHighWarning.fbrValue						(_usiParaNr := 18, itfConfigFb := fbConfigFile);
scParameter.scHighWarning.fbtDelayTillWarning			(_usiParaNr := 19, itfConfigFb := fbConfigFile);

(* High alarm *)
scParameter.scHighAlarm.fbxDoesAlarm					(_usiParaNr := 20, itfConfigFb := fbConfigFile);
scParameter.scHighAlarm.fbrValue						(_usiParaNr := 21, itfConfigFb := fbConfigFile);
scParameter.scHighAlarm.fbrHysterese					(_usiParaNr := 22, itfConfigFb := fbConfigFile);
scParameter.scHighAlarm.fbtDeleayTillAlarm				(_usiParaNr := 23, itfConfigFb := fbConfigFile);
scParameter.scHighAlarm.fbiTypeOfAcknolage				(_usiParaNr := 24, itfConfigFb := fbConfigFile, _MinInit := 0 , _MaxInit := 2);
scParameter.scHighAlarm.fbiRetryTillLock				(_usiParaNr := 25, itfConfigFb := fbConfigFile);

(* Alarm *)
scParameter.scAnalogAlarm.fbxEnableOverflowAl			(_usiParaNr := 26, itfConfigFb := fbConfigFile);
scParameter.scAnalogAlarm.fbxEnableUnderflowAl			(_usiParaNr := 27, itfConfigFb := fbConfigFile);

(* Alarm extra conditions *)
scParameter.scAlCondition.fbxEnable 					(_usiParaNr := 28, itfConfigFb := fbConfigFile);
scParameter.scAlCondition.fbtDelayTillCondition			(_usiParaNr := 29, itfConfigFb := fbConfigFile);

(* Alarm reset after... *)
scParameter.scAlarmReset.fbtDelayTillReset				(_usiParaNr := 30, itfConfigFb := fbConfigFile);

(* InfluxDb *)
scParameter.scInfluxDb.fbxEnable            			(_usiParaNr := 31, ItfConfigFb := fbconfigFile);

(* Visu *)
scParameter.scVisu.fbusiDezimalPos						(_usiParaNr := 32, ItfConfigFb := fbconfigFile, _minInit := 0, _maxInit := 3);

xConfigError := fbConfigFile.xError;
END_ACTION

PROPERTY P_scAnalogAlarm_fbxEnableOverflowAl : CtaSysConfig.ITF_DATATYPE
GET
P_scAnalogAlarm_fbxEnableOverflowAl:= scParameter.scAnalogAlarm.fbxEnableOverflowAl;
END_GET
END_PROPERTY

PROPERTY P_scAnalogAlarm_fbxEnableUnderflowAl : CtaSysConfig.ITF_DATATYPE
GET
P_scAnalogAlarm_fbxEnableUnderflowAl := scParameter.scAnalogAlarm.fbxEnableUnderflowAl;
END_GET
END_PROPERTY

PROPERTY P_scBase_fbxEnable : CtaSysConfig.ITF_DATATYPE
GET
P_scBase_fbxEnable := scParameter.scBase.fbxEnable;
END_GET
END_PROPERTY

PROPERTY P_scVisu_fbusiDezimalPos : CtaSysConfig.ITF_DATATYPE
GET
P_scVisu_fbusiDezimalPos := scParameter.scVisu.fbusiDezimalPos;
END_GET
END_PROPERTY

PROPERTY P_scAlCondition_fbxEnable : CtaSysConfig.ITF_DATATYPE
GET
P_scAlCondition_fbxEnable := scParameter.scAlCondition.fbxEnable;
END_GET
END_PROPERTY

PROPERTY P_scAlCondition_fbtDelayTillCondition : CtaSysConfig.ITF_DATATYPE
GET
P_scAlCondition_fbtDelayTillCondition := scParameter.scAlCondition.fbtDelayTillCondition;
END_GET
END_PROPERTY

PROPERTY P_scHighAlarm_fbiRetryTillLock : CtaSysConfig.ITF_DATATYPE
GET
P_scHighAlarm_fbiRetryTillLock := scParameter.scHighAlarm.fbiRetryTillLock;
END_GET
END_PROPERTY

PROPERTY P_scHighAlarm_fbiTypeOfAcknolage : CtaSysConfig.ITF_DATATYPE
GET
P_scHighAlarm_fbiTypeOfAcknolage := scParameter.scHighAlarm.fbiTypeOfAcknolage;
END_GET
END_PROPERTY

PROPERTY P_scHighAlarm_fbrHysterese : CtaSysConfig.ITF_DATATYPE
GET
P_scHighAlarm_fbrHysterese := scParameter.scHighAlarm.fbrHysterese;
END_GET
END_PROPERTY

PROPERTY P_scHighAlarm_fbrValue : CtaSysConfig.ITF_DATATYPE
GET
P_scHighAlarm_fbrValue := scParameter.scHighAlarm.fbrValue;
END_GET
END_PROPERTY

PROPERTY P_scHighAlarm_fbtDelayTillAlarm : CtaSysConfig.ITF_DATATYPE
GET
P_scHighAlarm_fbtDelayTillAlarm := scParameter.scHighAlarm.fbtDeleayTillAlarm;
END_GET
END_PROPERTY

PROPERTY P_scHighAlram_fbxDoesAlarm : CtaSysConfig.ITF_DATATYPE
GET
P_scHighAlram_fbxDoesAlarm := scParameter.scHighAlarm.fbxDoesAlarm;
END_GET
END_PROPERTY

PROPERTY P_scHighWarning_fbrValue : CtaSysConfig.ITF_DATATYPE
GET
P_scHighWarning_fbrValue := scParameter.scHighWarning.fbrValue;
END_GET
END_PROPERTY

PROPERTY P_scHighWarning_fbtDelayTillWarning : CtaSysConfig.ITF_DATATYPE
GET
P_scHighWarning_fbtDelayTillWarning := scParameter.scHighWarning.fbtDelayTillWarning;
END_GET
END_PROPERTY

PROPERTY P_scHighWarning_fbxDoesWarning : CtaSysConfig.ITF_DATATYPE
GET
P_scHighWarning_fbxDoesWarning := scParameter.scHighWarning.fbxDoesWarning;
END_GET
END_PROPERTY

PROPERTY P_scInfluxDb_fbxEnable : CtaSysConfig.ITF_DATATYPE
GET
P_scInfluxDb_fbxEnable := scParameter.scInfluxDb.fbxEnable;
END_GET
END_PROPERTY

PROPERTY P_scLoAlarm_fbiRetryTillLock : CtaSysConfig.ITF_DATATYPE
GET
P_scLoAlarm_fbiRetryTillLock := scParameter.scLoAlarm.fbiRetryTillLock;
END_GET
END_PROPERTY

PROPERTY P_scLoAlarm_fbiTypeOfAcknolage : CtaSysConfig.ITF_DATATYPE
GET
P_scLoAlarm_fbiTypeOfAcknolage := scParameter.scLoAlarm.fbiTypeOfAcknolage;
END_GET
END_PROPERTY

PROPERTY P_scLoAlarm_fbrHysterese : CtaSysConfig.ITF_DATATYPE
GET
P_scLoAlarm_fbrHysterese := scParameter.scLoAlarm.fbrHysterese;
END_GET
END_PROPERTY

PROPERTY P_scLoAlarm_fbrValue : CtaSysConfig.ITF_DATATYPE
GET
P_scLoAlarm_fbrValue := scParameter.scLoAlarm.fbrValue;
END_GET
END_PROPERTY

PROPERTY P_scLoAlarm_fbtDelayTillAlarm : CtaSysConfig.ITF_DATATYPE
GET
P_scLoAlarm_fbtDelayTillAlarm := scParameter.scLoAlarm.fbtDeleayTillAlarm;
END_GET
END_PROPERTY

PROPERTY P_scLoAlarm_fbxDoesAlarm : CtaSysConfig.ITF_DATATYPE
GET
P_scLoAlarm_fbxDoesAlarm := scParameter.scLoAlarm.fbxDoesAlarm;
END_GET
END_PROPERTY

PROPERTY P_scLoWarning_fbrValue : CtaSysConfig.ITF_DATATYPE
GET
P_scLoWarning_fbrValue := scParameter.scLoWarning.fbrValue;
END_GET
END_PROPERTY

PROPERTY P_scLoWarning_fbtDelayTillWarning : CtaSysConfig.ITF_DATATYPE
GET
P_scLoWarning_fbtDelayTillWarning := scParameter.scLoWarning.fbtDelayTillWarning;
END_GET
END_PROPERTY

PROPERTY P_scLoWarning_fbxDoesWarning : CtaSysConfig.ITF_DATATYPE
GET
P_scLoWarning_fbxDoesWarning := scParameter.scLoWarning.fbxDoesWarning;
END_GET
END_PROPERTY

PROPERTY P_scManual_fbrManualOnY : CtaSysConfig.ITF_DATATYPE
GET
P_scManual_fbrManualOnY := scParameter.scManual.fbrManualOnY;
END_GET
END_PROPERTY

PROPERTY P_scManual_fbuiManualControl : CtaSysConfig.ITF_DATATYPE
GET
P_scManual_fbuiManualControl := scParameter.scManual.fbuiManualControl;
END_GET
END_PROPERTY

PROPERTY P_scManual_fbuiManualState : CtaSysConfig.ITF_DATATYPE
GET
P_scManual_fbuiManualState := scParameter.scManual.fbuiManualState;
END_GET
END_PROPERTY

PROPERTY P_scManual_fbxAllowManualOn : CtaSysConfig.ITF_DATATYPE
GET
P_scManual_fbxAllowManualOn := scParameter.scManual.fbxAlowManualOn;
END_GET
END_PROPERTY

PROPERTY P_scAlarmReset_fbtDealyTillReset : CtaSysConfig.ITF_DATATYPE
GET
P_scAlarmReset_fbtDealyTillReset := scParameter.scAlarmReset.fbtDelayTillReset;
END_GET
END_PROPERTY

PROPERTY P_scFilter_fbrValue : CtaSysConfig.ITF_DATATYPE
GET
P_scFilter_fbrValue := scParameter.scFilter.fbrValue;
END_GET
END_PROPERTY

PROPERTY P_scFilter_fbxEnabled : CtaSysConfig.ITF_DATATYPE
GET
P_scFilter_fbxEnabled := scParameter.scFilter.fbxEnabled;
END_GET
END_PROPERTY

PROPERTY proSensorITF : CtaSysIO.ITF_IO;
GET
proSensorITF := ITF_IO_IN;
END_GET
END_PROPERTY

PROPERTY proRawValue : STRING
GET
IF xIsITF THEN
	IF __QUERYINTERFACE (_ITF_DI,_ITF_DI) THEN	
		proRawValue := TO_STRING(_ITF_DI.proValue);
	ELSIF __QUERYINTERFACE(_ITF_AI,_ITF_AI) THEN
		IF _ITF_AI.proModuleType = CtaSysIO.enModuleType.DC_0_10V_IN THEN
			proRawValue :=	CONCAT(TO_STRING(_ITF_AI.proPhysicalValue),' v');
		ELSIF _ITF_AI.proModuleType = CtaSysIO.enModuleType.DC_4_20mA_IN THEN
			proRawValue :=	CONCAT(TO_STRING(_ITF_AI.proPhysicalValue),' mA');
		ELSIF _ITF_AI.proModuleType = CtaSysIO.enModuleType.ohm THEN
			proRawValue :=	CONCAT(TO_STRING(_ITF_AI.proPhysicalValue),' °C');
		ELSE
			proRawValue := '';	
		END_IF
	ELSE
		proRawValue := '';			
	END_IF	
ELSIF xIsBool THEN
	proRawValue := TO_STRING(xValueIn);
ELSIF xIsReal THEN
	proRawValue := TO_STRING(rValueIn);
ELSE
	proRawValue := '';	
END_IF
END_GET
END_PROPERTY

//FB_Init ist immer implizit verfügbar und wird primär für die Initialisierung verwendet.
//Der Rückgabewert wird nicht ausgewertet. Für gezielte Einflussnahme können Sie
//die Methoden explizit deklarieren und darin mit dem Standard-Initialisierungscode 
//zusätzlichen Code bereitstellen. Sie können den Rückgabewert auswerten.
METHOD FB_INIT: BOOL
VAR_INPUT    
bInitRetains: BOOL; // TRUE: Die Retain-Variablen werden initialisiert (Reset warm / Reset kalt)    
bInCopyCode: BOOL;  // TRUE: Die Instanz wird danach in den Kopiercode kopiert (Online-Change)
END_VAR
VAR
    ITF_SENSOR_THIS             :   ITF_SENSOR;
    ITF_SENSOR_QUERRY           :   ITF_SENSOR;
END_VAR
IF NOT bInCopyCode THEN
    ITF_SENSOR_THIS := THIS^;
    IF __QUERYINTERFACE(ITF_SENSOR_THIS,ITF_SENSOR_QUERRY) THEN
        diArrayPosition := GVL_SENSOR.fbSensor_Collector.metRegistry(ITF_SENSOR_QUERRY);
    END_IF;
END_IF;
END_METHOD

PROPERTY proSoftwareValue : STRING
GET
IF xIsBool OR ( xIsITF AND __QUERYINTERFACE (_ITF_DI,_ITF_DI)) THEN
	proSoftwareValue := TO_STRING(xValue);
ELSIF xIsReal THEN
	proSoftwareValue := CONCAT(TO_STRING(CTASYsCONFIG.fcRealToString(rValue,scparameter.scVisu.fbusiDezimalPos.usiValue)),stAlternateUnit);	 
ELSIF xIsITF AND __QUERYINTERFACE(_ITF_AI,_ITF_AI) THEN
	IF _ITF_AI.proModuleType = CtaSysIO.enModuleType.OHM THEN
		proSoftwareValue := CONCAT(TO_STRING(CTASYsCONFIG.fcRealToString(rValue,scparameter.scVisu.fbusiDezimalPos.usiValue)),'°C') ;
	ELSE
		proSoftwareValue := CONCAT(TO_STRING(CTASYsCONFIG.fcRealToString(rValue,scparameter.scVisu.fbusiDezimalPos.usiValue)),CtaSysConfig.fcGetValueFromDataType(_ITF_AI.P_scfbAI_fbstPhysicalUnit)) ;
	END_IF	
ELSE
	proSoftwareValue := '';
END_IF
END_GET
END_PROPERTY

PROPERTY proIsWarning : BOOL
GET
proIsWarning := xIsWarning;
END_GET
END_PROPERTY

PROPERTY proIsHandOnOrOff : BOOL
GET
proIsHandOnOrOff := xIsHand;
END_GET
END_PROPERTY

PROPERTY proIsReady : BOOL
GET
proIsReady := xIsEnabled AND NOT xIsError;
END_GET
END_PROPERTY

PROPERTY proHandOff : BOOL
SET
IF proHandOff THEN
	scParameter.scManual.fbuiManualState.proValue := 1;
END_IF
END_SET
GET
proHandOff := xIsHandOff;
END_GET
END_PROPERTY

PROPERTY proHandOn : BOOL
GET
proHandOn := xIsHandOn OR xIsHandMode;
END_GET
SET
IF proHandOn THEN
	scParameter.scManual.fbuiManualState.proValue := 2;
END_IF
END_SET
END_PROPERTY

PROPERTY proHandOnY : REAL
SET
scParameter.scManual.fbrManualOnY.proValue := proHandOnY;
END_SET
GET
proHandOnY := scParameter.scManual.fbrManualOnY.proValue;
END_GET
END_PROPERTY

PROPERTY proAuto : BOOL
SET
IF proAuto THEN
	scParameter.scManual.fbuiManualState.provalue := 0;
END_IF
END_SET
GET
proAuto := xIsAuto;
END_GET
END_PROPERTY

PROPERTY proManualTrue : BOOL
SET
IF proManualTrue THEN
	scParameter.scManual.fbuiManualControl.proValue := 1;
END_IF
END_SET
GET
proManualTrue := xManualValue;
END_GET
END_PROPERTY

PROPERTY proManualFalse : BOOL
SET
IF proManualFalse THEN
	scParameter.scManual.fbuiManualControl.proValue := 0;
END_IF
END_SET
GET
proManualFalse := NOT xManualValue;
END_GET
END_PROPERTY

PROPERTY proValueInputType : enInputType
GET
proValueInputType := enValueInputType;
END_GET
END_PROPERTY

METHOD metSetITF
VAR_INPUT
	ITF_IN		:	CtaSysIO.ITF_IO;
END_VAR
ITF_IO_IN := ITF_IN;
xIsITF 	:= TRUE;
xIsBool := FALSE;
xIsReal := FALSE;
END_METHOD

ACTION actDigital:
IF _ITF_DI <> 0 THEN
	xValueTemp := _ITF_DI.proValue;
ELSE
	xValueTemp := xValueIn;	
END_IF

(* Low Controll *)
xLoWarning      := fcLowControl(xEn   := scParameter.scLoWarning.fbxDoesWarning.proValue,
								rIst  := TO_REAL(xValueTemp),
								rLow  := 0,
								rHyst := 0,
								xTrig := 0);
								
xLoAlarm      	:= fcLowControl(xEn   := scParameter.scLoAlarm.fbxDoesAlarm.proValue,
								rIst  := TO_REAL(xValueTemp),
								rLow  := 0,
								rHyst := 0,
								xTrig := 0);

(* High Controll *)
xHiWarning     := fcHighControl(xEn   := scParameter.scHighWarning.fbxDoesWarning.proValue,
								rIst  := TO_REAL(xValueTemp),
								rHigh := 1,
								rHyst := 0,
								xTrig := 0);
								
xHiAlarm       := fcHighControl(xEn   := scParameter.scHighAlarm.fbxDoesAlarm.proValue,
								rIst  := TO_REAL(xValueTemp),
								rHigh := 1,
								rHyst := 0,
								xTrig := 0);

(* Hand Off *)
IF scParameter.scManual.fbuiManualState.proValue = 1 THEN
	xValue := NOT xValueTemp;	
	xIsHandMode := FALSE;
(* Hand On *)	
ELSIF scParameter.scManual.fbuiManualState.proValue <> 2 AND NOT xEnHandMode THEN
	(* Value *)
	xValue := xValueTemp;
	xIsHandMode := FALSE;
ELSE
	xValue := SEL(xEnHandMode,xManualValue,TO_BOOL(rSimValue));
	xIsHandMode := TRUE;
	
	IF NOT scParameter.scManual.fbxAlowManualOn.proValue AND NOT xEnHandMode THEN
		xValue := xValueTemp;
		xIsHandMode := FALSE;
	END_IF
END_IF

rValue := TO_REAL(xValue);
END_ACTION

ACTION actAnalog:
IF _ITF_AI <> 0 THEN	
	rValueUngefiltert      := _ITF_AI.proValue;
	xOk					   := _ITF_AI.proOK; 
ELSE	
	rValueUngefiltert      := rValueIn; 
END_IF
        
(* Low Controll *)
xLoWarning	:= fcLowControl(xEn   := scParameter.scLoWarning.fbxDoesWarning.proValue,
							rIst  := rValueUngefiltert,
							rLow  := scParameter.scLoWarning.fbrValue.proValue,
							rHyst := 0,
							xTrig := 0);
(* ToLow Controll *)
xLoAlarm    := fcLowControl(xEn   := scParameter.scLoAlarm.fbxDoesAlarm.proValue,
							rIst  := rValueUngefiltert,
							rlow  := scParameter.scLoAlarm.fbrValue.proValue,
							rHyst := scParameter.scLoAlarm.fbrHysterese.proValue,
							xTrig := xLoAlarm);
							
(* High Controll *)
xHiWarning := fcHighControl(xEn   := scParameter.scHighWarning.fbxDoesWarning.proValue,
							rIst  := rValueUngefiltert,
							rHigh := scParameter.scHighWarning.fbrValue.proValue,
							rHyst := 0,
							xTrig := 0);
(* ToHigh Controll *)
xHiAlarm   := fcHighControl(xEn   := scParameter.scHighAlarm.fbxDoesAlarm.proValue,
							rIst  := rValueUngefiltert,
							rHigh := scParameter.scHighAlarm.fbrValue.proValue,
							rHyst := scParameter.scHighAlarm.fbrHysterese.proValue,
							xTrig := xHiAlarm);
							
(* Filter *)
IF scParameter.scFilter.fbxEnabled.proValue THEN
	fbFilter   				   (rIn  	:= rValueUngefiltert,
								rFilter := scParameter.scFilter.fbrValue.proValue);
	(* Value Out*)
	rValueTemp  := fbFilter.rOut;
ELSE
	(* Value Out*)
	rValueTemp  := rValueUngefiltert;
END_IF

IF scParameter.scManual.fbuiManualState.proValue = 1 THEN
	rValue := 0;
	xIsHandMode := FALSE;
ELSIF scParameter.scManual.fbuiManualState.proValue <> 2 AND NOT xEnHandMode THEN
	rValue := rValueTemp;
	xIsHandMode := FALSE;
ELSE
	rValue := SEL(xEnHandMode,scParameter.scManual.fbrManualOnY.proValue,rSimValue);
	xIsHandMode := TRUE;
	
	IF NOT scParameter.scManual.fbxAlowManualOn.proValue AND NOT xEnHandMode THEN
		rValue := rValueTemp;
		xIsHandMode := FALSE;
	END_IF
END_IF

xValue  := scEWI.iError = 0 AND SEL(_ITF_AI <> 0,TRUE ,xOk);
END_ACTION

PROPERTY proPhysicalValue : STRING
GET
IF xIsITF THEN
	IF __QUERYINTERFACE (_ITF_AI,_ITF_AI)THEN
		proPhysicalValue := CONCAT(TO_STRING(_ITF_AI.proValue),CtaSysConfig.fcGetValueFromDataType(_ITF_AI.P_scfbAI_fbstPhysicalUnit));
	ELSIF __QUERYINTERFACE (_ITF_DI,_ITF_DI) THEN
		proPhysicalValue := TO_STRING(_ITF_DI.proValue);
	ELSE
		proPhysicalValue := '';
	END_IF
ELSIF xIsBool THEN
	proPhysicalValue := TO_STRING(xValueIn);
ELSIF xIsReal THEN
	proPhysicalValue :=TO_STRING(rValueIn);
ELSE
	proPhysicalValue := '';
END_IF
END_GET
END_PROPERTY

ACTION actReCalculate:
IF __QUERYINTERFACE(ITF_RC_QUERY,ITF_RC_QUERY) THEN
	ITF_RC_QUERY.VALUE := rValue;
	rValueRC := ITF_RC_QUERY.CALCULATET_VALUE;
ELSE
	rValueRC := rValue;
END_IF;
END_ACTION

PROPERTY ITF_RC : CtaSysSensorReCalculation.ITF_SENSOR_RE_CALCULATE
SET
ITF_RC_QUERY := ITF_RC;
END_SET
GET
ITF_RC := ITF_RC_QUERY;
END_GET
END_PROPERTY

ACTION actMbState:
IF NOT xModbusTest THEN
    (* State Word 0 Digital Info*)
    ayMbStateWord[0].00     := xValue;
    ayMbStateWord[0].01     := FALSE;
    ayMbStateWord[0].02     := FALSE;
    ayMbStateWord[0].03     := FALSE;
    ayMbStateWord[0].04     := FALSE;
    ayMbStateWord[0].05     := FALSE;
    ayMbStateWord[0].06     := FALSE;
    ayMbStateWord[0].07     := FALSE;
    ayMbStateWord[0].08     := xIsHand;
    ayMbStateWord[0].09     := xIsAuto;
    ayMbStateWord[0].10     := FALSE;
    ayMbStateWord[0].11     := FALSE;
    ayMbStateWord[0].12     := FALSE;
    ayMbStateWord[0].13     := FALSE;
    ayMbStateWord[0].14     := xIsWarning;
    ayMbStateWord[0].15     := xIsError;
	
	IF (enValueInputType = enInputType.DigitalInput) OR (enValueInputType = enInputType.Digital_ITF_Input) THEN
		(* State Word 1 setpoint*)
		ayMbStateWord[1]   	:= TO_WORD(TO_INT(xValue));
		(* State Word 2 actual value*)
		ayMbStateWord[3]	:= TO_WORD(TO_INT(xValue));
	ELSE
		 (* State Word 1 setpoint*)
		ayMbStateWord[1]   	:= TO_WORD(TO_INT(rValue * 10));
		(* State Word 2 actual value*)
		ayMbStateWord[2]	:= TO_WORD(TO_INT(rValueRC * 10));
		(* State Word 3 actual value*)
		ayMbStateWord[3]	:=	SEL(enValueInputType = enInputType.Analog_ITF_Input,TO_WORD(TO_INT(rValue * 10)),TO_WORD(TO_INT(_ITF_AI.proPhysicalValue * 10)));	
	END_IF
END_IF;
END_ACTION

PROPERTY proModbusTest : BOOL
SET
xModbusTest := proModbusTest;
END_SET
GET
proModbusTest := xModbusTest;
END_GET
END_PROPERTY

{warning disable C0410}
PROPERTY proModbusStateWord : REFERENCE TO ARRAY[0..3] OF WORD
{warning restore C0410}
GET
proModbusStateWord REF= ayMbStateWord;
END_GET
END_PROPERTY

{warning disable C0410}
PROPERTY proModbusControllWord : REFERENCE TO ARRAY[0..3] OF WORD
{warning restore C0410}
GET
proModbusControllWord REF= ayMbControllWord;
END_GET
END_PROPERTY

PROPERTY prorValue : REAL
GET
prorValue := rValue;
END_GET
END_PROPERTY

END_FUNCTION_BLOCK

// 30 Program Organization Units/Abstracte Bausteine/fbSensorTabellenInfo
{attribute 'hide'} 
FUNCTION_BLOCK INTERNAL ABSTRACT fbSensorTabellenInfo EXTENDS CtaAppBmk.fbBMK IMPLEMENTS ITF_SENSOR_TABELLE_INFO

PROPERTY proStateSymbol : STRING
GET
END_GET
END_PROPERTY

PROPERTY proSoftwareValue : STRING
GET
END_GET
END_PROPERTY

PROPERTY proRawValue : STRING
GET
END_GET
END_PROPERTY

PROPERTY proEnSymbol : STRING
GET
END_GET
END_PROPERTY

PROPERTY proPhysicalValue : STRING
GET
END_GET
END_PROPERTY

END_FUNCTION_BLOCK

// 21 Interface/ITF_SENSOR_TABELLE_INFO
INTERFACE INTERNAL ITF_SENSOR_TABELLE_INFO EXTENDS CtaAppBmk.ITF_BMK

PROPERTY proRawValue : STRING
GET
END_GET
END_PROPERTY

PROPERTY proSoftwareValue : STRING
GET
END_GET
END_PROPERTY

{attribute 'hide'} 
PROPERTY INTERNAL proEnSymbol : STRING
GET
END_GET
END_PROPERTY

{attribute 'hide'} 
PROPERTY INTERNAL proStateSymbol : STRING
GET
END_GET
END_PROPERTY

PROPERTY proPhysicalValue : STRING
GET
END_GET
END_PROPERTY

END_INTERFACE

// 21 Interface/ITF_SENSOR
INTERFACE ITF_SENSOR EXTENDS ITF_SENSOR_TABELLE_INFO , CtaAppModbusSpezifikation.ITF_MODBUS_SPEZIFIKATION

{attribute 'hide'} 
PROPERTY proConfigError : BOOL
GET
END_GET
END_PROPERTY

PROPERTY P_scBase_fbxEnable : CtaSysConfig.ITF_DATATYPE
GET
END_GET
END_PROPERTY

PROPERTY P_scVisu_fbusiDezimalPos : CtaSysConfig.ITF_DATATYPE
GET
END_GET
END_PROPERTY

PROPERTY P_scManual_fbxAllowManualOn : CtaSysConfig.ITF_DATATYPE
GET
END_GET
END_PROPERTY

PROPERTY P_scManual_fbuiManualState : CtaSysConfig.ITF_DATATYPE
GET
END_GET
END_PROPERTY

PROPERTY P_scManual_fbuiManualControl : CtaSysConfig.ITF_DATATYPE
GET
END_GET
END_PROPERTY

PROPERTY P_scManual_fbrManualOnY : CtaSysConfig.ITF_DATATYPE
GET
END_GET
END_PROPERTY

PROPERTY P_scFilter_fbxEnabled : CtaSysConfig.ITF_DATATYPE
GET
END_GET
END_PROPERTY

PROPERTY P_scFilter_fbrValue : CtaSysConfig.ITF_DATATYPE
GET
END_GET
END_PROPERTY

PROPERTY P_scLoWarning_fbxDoesWarning : CtaSysConfig.ITF_DATATYPE
GET
END_GET
END_PROPERTY

PROPERTY P_scLoWarning_fbrValue : CtaSysConfig.ITF_DATATYPE
GET
END_GET
END_PROPERTY

PROPERTY P_scLoWarning_fbtDelayTillWarning : CtaSysConfig.ITF_DATATYPE
GET
END_GET
END_PROPERTY

PROPERTY P_scLoAlarm_fbxDoesAlarm : CtaSysConfig.ITF_DATATYPE
GET
END_GET
END_PROPERTY

PROPERTY P_scLoAlarm_fbrValue : CtaSysConfig.ITF_DATATYPE
GET
END_GET
END_PROPERTY

PROPERTY P_scLoAlarm_fbrHysterese : CtaSysConfig.ITF_DATATYPE
GET
END_GET
END_PROPERTY

PROPERTY P_scLoAlarm_fbtDelayTillAlarm : CtaSysConfig.ITF_DATATYPE
GET
END_GET
END_PROPERTY

PROPERTY P_scLoAlarm_fbiRetryTillLock : CtaSysConfig.ITF_DATATYPE
GET
END_GET
END_PROPERTY

PROPERTY P_scLoAlarm_fbiTypeOfAcknolage : CtaSysConfig.ITF_DATATYPE
GET
END_GET
END_PROPERTY

PROPERTY P_scHighWarning_fbxDoesWarning : CtaSysConfig.ITF_DATATYPE
GET
END_GET
END_PROPERTY

PROPERTY P_scHighWarning_fbrValue : CtaSysConfig.ITF_DATATYPE
GET
END_GET
END_PROPERTY

PROPERTY P_scHighWarning_fbtDelayTillWarning : CtaSysConfig.ITF_DATATYPE
GET
END_GET
END_PROPERTY

PROPERTY P_scHighAlram_fbxDoesAlarm : CtaSysConfig.ITF_DATATYPE
GET
END_GET
END_PROPERTY

PROPERTY P_scHighAlarm_fbrValue : CtaSysConfig.ITF_DATATYPE
GET
END_GET
END_PROPERTY

PROPERTY P_scHighAlarm_fbrHysterese : CtaSysConfig.ITF_DATATYPE
GET
END_GET
END_PROPERTY

PROPERTY P_scHighAlarm_fbtDelayTillAlarm : CtaSysConfig.ITF_DATATYPE
GET
END_GET
END_PROPERTY

PROPERTY P_scHighAlarm_fbiRetryTillLock : CtaSysConfig.ITF_DATATYPE
GET
END_GET
END_PROPERTY

PROPERTY P_scHighAlarm_fbiTypeOfAcknolage : CtaSysConfig.ITF_DATATYPE
GET
END_GET
END_PROPERTY

PROPERTY P_scInfluxDb_fbxEnable : CtaSysConfig.ITF_DATATYPE
GET
END_GET
END_PROPERTY

PROPERTY P_scAnalogAlarm_fbxEnableOverflowAl : CtaSysConfig.ITF_DATATYPE
GET
END_GET
END_PROPERTY

PROPERTY P_scAnalogAlarm_fbxEnableUnderflowAl : CtaSysConfig.ITF_DATATYPE
GET
END_GET
END_PROPERTY

PROPERTY P_scAlCondition_fbxEnable : CtaSysConfig.ITF_DATATYPE
GET
END_GET
END_PROPERTY

PROPERTY P_scAlCondition_fbtDelayTillCondition : CtaSysConfig.ITF_DATATYPE
GET
END_GET
END_PROPERTY

PROPERTY P_scAlarmReset_fbtDealyTillReset : CtaSysConfig.ITF_DATATYPE
GET
END_GET
END_PROPERTY

PROPERTY proSensorITF : CtaSysIO.ITF_IO;
GET
END_GET
END_PROPERTY

{attribute 'hide'} 
PROPERTY INTERNAL proCountedError : INT
GET
END_GET
END_PROPERTY

{attribute 'hide'} 
PROPERTY INTERNAL proCountedInfo : INT
GET
END_GET
END_PROPERTY

{attribute 'hide'} 
PROPERTY INTERNAL proITF_REPORTMANAGER : CtaAppReport.ITF_REPORTMANAGER
GET
END_GET
END_PROPERTY

{attribute 'hide'} 
PROPERTY INTERNAL proCountedWarning : INT
GET
END_GET
END_PROPERTY

PROPERTY proIsHandOnOrOff : BOOL
GET
END_GET
END_PROPERTY

PROPERTY proHandOn : BOOL
SET
END_SET
GET
END_GET
END_PROPERTY

PROPERTY proIsError : BOOL
GET
END_GET
END_PROPERTY

PROPERTY proIsWarning : BOOL
GET
END_GET
END_PROPERTY

PROPERTY proEn : BOOL
GET
END_GET
SET
END_SET
END_PROPERTY

PROPERTY proIsEnabled : BOOL
GET
END_GET
END_PROPERTY

PROPERTY proHandOff : BOOL
SET
END_SET
GET
END_GET
END_PROPERTY

PROPERTY proHandOnY : REAL
SET
END_SET
GET
END_GET
END_PROPERTY

PROPERTY proIsReady : BOOL
GET
END_GET
END_PROPERTY

PROPERTY proAuto : BOOL
SET
END_SET
GET
END_GET
END_PROPERTY

PROPERTY proManualFalse : BOOL
SET
END_SET
GET
END_GET
END_PROPERTY

PROPERTY proManualTrue : BOOL
SET
END_SET
GET
END_GET
END_PROPERTY

PROPERTY proValueInputType : enInputType
GET
END_GET
END_PROPERTY

PROPERTY proxErrorConditionValue : BOOL;
GET
END_GET
END_PROPERTY

PROPERTY proInvertierung : BOOL
GET
END_GET
END_PROPERTY

PROPERTY prorValue : REAL
GET
END_GET
END_PROPERTY

{attribute 'monitoring' := 'variable'}
PROPERTY proLockDown : BOOL
GET
END_GET
END_PROPERTY

{attribute 'monitoring' := 'variable'}
PROPERTY proAvailable : BOOL
GET
END_GET
END_PROPERTY

{attribute 'monitoring' := 'variable'}
PROPERTY proAcknowlege : BOOL
GET
END_GET
END_PROPERTY

PROPERTY proAtIconNr : UINT
GET
END_GET
SET
END_SET
END_PROPERTY

PROPERTY ITF_RC : CtaSysSensorReCalculation.ITF_SENSOR_RE_CALCULATE
SET
END_SET
GET
END_GET
END_PROPERTY

{warning disable C0410}
PROPERTY proModbusStateWord : REFERENCE TO ARRAY[0..3] OF WORD
{warning restore C0410}
GET
END_GET
END_PROPERTY

{attribute 'hide'} 
PROPERTY INTERNAL proModbusTest : BOOL
GET
END_GET
SET
END_SET
END_PROPERTY

{warning disable C0410}
PROPERTY proModbusControllWord : REFERENCE TO ARRAY[0..3] OF WORD
{warning restore C0410}
GET
END_GET
END_PROPERTY

END_INTERFACE

// 30 Program Organization Units/fb's/Collector/fbSensor_Collector
FUNCTION_BLOCK fbSensor_Collector IMPLEMENTS ITF_SENSOR_COLLECTOR
VAR_INPUT
END_VAR
VAR_OUTPUT
END_VAR
VAR
    ayAT_INTERFACE          : ARRAY[1..Parameter.iMaxSensor] OF ITF_SENSOR;   
    ayAT_INTERFACE_SORTET   : ARRAY[1..Parameter.iMaxSensor] OF ITF_SENSOR; 
    xIsSortet               : BOOL;
    diNext                  : DINT    := 1;
    diMin                   : DINT    := 1;
    diMax                   : DINT;
    diMaxSort               : DINT;
    xError                  : BOOL;
    xBufferError            : BOOL;
    diMissedBuffer          : DINT;
END_VAR

METHOD metRegistry : DINT
VAR_INPUT
    ITF_AT_IN   :   ITF_SENSOR;
END_VAR
VAR
    diArrayPos  :   DINT;
    diCount     :   DINT;
END_VAR
IF ITF_AT_IN <> 0 THEN
    diArrayPos := __XADD(ADR(diNext),1);
    IF diArrayPos <= Parameter.iMaxSensor AND diArrayPos >= 1 THEN
        IF __QUERYINTERFACE(ITF_AT_IN,ayAT_INTERFACE[diArrayPos]) THEN
            metRegistry             := diArrayPos;
            GVL_SENSOR.xValidData       := TRUE;
            diCount    := __XADD(ADR(diMax),1);
        END_IF;
    ELSE
        IF diArrayPos > Parameter.iMaxSensor THEN
            xBufferError := TRUE;
            diMissedBuffer := diArrayPos - Parameter.iMaxSensor;
		END_IF;
        xError      := TRUE; 
        metRegistry := 0;
    END_IF;   
ELSE
    xError := TRUE; 
    metRegistry := 0;
END_IF;
END_METHOD

PROPERTY proMin : INT
GET
proMin := 1;
END_GET
END_PROPERTY

PROPERTY proMax : UINT
GET
IF xIsSortet THEN
    proMax := LIMIT(0,TO_UINT(diMaxSort),65535);    
ELSE
    proMax := LIMIT(0,TO_UINT(diMax),65535);    
END_IF
END_GET
END_PROPERTY

PROPERTY proaySensorTabelle : ARRAY[1..Parameter.iMaxSensor] OF ITF_SENSOR_TABELLE_INFO
GET
VAR
    diFor   :   DINT;
END_VAR
IF xIsSortet THEN
    FOR diFor := LOWER_BOUND(proaySensorTabelle,1) TO UPPER_BOUND(proaySensorTabelle,1) DO
        __QUERYINTERFACE(ayAT_INTERFACE_SORTET[diFor],proaySensorTabelle[diFor]);   
	END_FOR
ELSE
    FOR diFor := LOWER_BOUND(proaySensorTabelle,1) TO UPPER_BOUND(proaySensorTabelle,1) DO
        __QUERYINTERFACE(ayAT_INTERFACE[diFor],proaySensorTabelle[diFor]);   
	END_FOR
END_IF;
END_GET
END_PROPERTY

PROPERTY proMissedBuffer : DINT
GET
proMissedBuffer := diMissedBuffer;
END_GET
END_PROPERTY

PROPERTY proBufferError : BOOL
GET
proBufferError := xBufferError;
END_GET
END_PROPERTY

PROPERTY proayAntrieb : ARRAY[1..Parameter.iMaxSensor] OF ITF_SENSOR
GET
VAR
    diFor   :   DINT;
END_VAR
IF xIsSortet THEN
    proayAntrieb := ayAT_INTERFACE_SORTET;
ELSE
    proayAntrieb := ayAT_INTERFACE;
END_IF;
END_GET
END_PROPERTY

METHOD metSortArray
VAR_INPUT
    stSearch    :   STRING;
    uiSort      :   UINT;
END_VAR
VAR
    diFor1      :   DINT;
    diFor2      :   DINT;
    diFill      :   DINT;
    ITF_AT_Temp :   ITF_SENSOR;    
    iBigger     :   INT;
END_VAR
IF stSearch <> '' THEN
    diMaxSort   := 0;
    diFill      := LOWER_BOUND(ayAT_INTERFACE,1); 
    FOR diFor1 := LOWER_BOUND(ayAT_INTERFACE,1) TO UPPER_BOUND(ayAT_INTERFACE,1) DO
        IF ayAT_INTERFACE[diFor1] <> 0 THEN
            IF FIND(ayAT_INTERFACE[diFor1].proGetBMK,stSearch) <> 0 OR FIND(ayAT_INTERFACE[diFor1].proGetVendorDesignation,stSearch) <> 0 THEN
                ayAT_INTERFACE_SORTET[diFill] := ayAT_INTERFACE[diFor1];
                diFill      := diFill + 1; 
                diMaxSort   := diFill -1; 
            END_IF;
        END_IF;
	END_FOR;
ELSE
    ayAT_INTERFACE_SORTET := ayAT_INTERFACE;
    diMaxSort := diMax;
END_IF; 
// 1 = Sort BMK
IF uiSort = 1 THEN
    FOR diFor1 := LOWER_BOUND(ayAT_INTERFACE_SORTET,1) TO diMaxSort DO 
        FOR diFor2 := LOWER_BOUND(ayAT_INTERFACE_SORTET,1) TO diMaxSort -1 DO 
            IF ayAT_INTERFACE_SORTET[diFor2] <> 0 AND ayAT_INTERFACE_SORTET[diFor2 + 1] <> 0 THEN
                IF LEN(ayAT_INTERFACE_SORTET[diFor2].proGetBMK) > LEN(ayAT_INTERFACE_SORTET[diFor2 + 1].proGetBMK) THEN
                    ITF_AT_Temp                         := ayAT_INTERFACE_SORTET[diFor2];
                    ayAT_INTERFACE_SORTET[diFor2]       := ayAT_INTERFACE_SORTET[diFor2 + 1];
                    ayAT_INTERFACE_SORTET[diFor2 + 1]   := ITF_AT_Temp; 
                ELSIF LEN(ayAT_INTERFACE_SORTET[diFor2].proGetBMK) = LEN(ayAT_INTERFACE_SORTET[diFor2 + 1].proGetBMK) THEN
                    iBigger := fcGetBigerStringValue(ayAT_INTERFACE_SORTET[diFor2].proGetBMK,ayAT_INTERFACE_SORTET[diFor2 + 1].proGetBMK);
                    IF iBigger = 1 THEN
                        ITF_AT_Temp                         := ayAT_INTERFACE_SORTET[diFor2];
                        ayAT_INTERFACE_SORTET[diFor2]       := ayAT_INTERFACE_SORTET[diFor2 + 1];
                        ayAT_INTERFACE_SORTET[diFor2 + 1]   := ITF_AT_Temp;                                                
					END_IF;
				END_IF;
            END_IF;       
        END_FOR;      
    END_FOR;     
// 2 = Sort Vendor Name    
ELSIF uiSort = 2 THEN
    FOR diFor1 := LOWER_BOUND(ayAT_INTERFACE_SORTET,1) TO diMaxSort DO 
        FOR diFor2 := LOWER_BOUND(ayAT_INTERFACE_SORTET,1) TO diMaxSort -1 DO 
            IF ayAT_INTERFACE_SORTET[diFor2] <> 0 AND ayAT_INTERFACE_SORTET[diFor2 + 1] <> 0 THEN
                iBigger := fcGetBigerStringValue(ayAT_INTERFACE_SORTET[diFor2].proGetVendorDesignation,ayAT_INTERFACE_SORTET[diFor2 + 1].proGetVendorDesignation);
                IF iBigger = 1 THEN
                    ITF_AT_Temp                         := ayAT_INTERFACE_SORTET[diFor2];
                    ayAT_INTERFACE_SORTET[diFor2]       := ayAT_INTERFACE_SORTET[diFor2 + 1];
                    ayAT_INTERFACE_SORTET[diFor2 + 1]   := ITF_AT_Temp;                                            
                END_IF;
            END_IF;       
        END_FOR;      
    END_FOR;
// 3 & 4 = Sort State  
ELSIF uiSort = 3 OR uiSort = 4 THEN
    FOR diFor1 := LOWER_BOUND(ayAT_INTERFACE_SORTET,1) TO diMaxSort DO 
        FOR diFor2 := LOWER_BOUND(ayAT_INTERFACE_SORTET,1) TO diMaxSort -1 DO 
            IF ayAT_INTERFACE_SORTET[diFor2] <> 0 AND ayAT_INTERFACE_SORTET[diFor2 + 1] <> 0 THEN
                IF ayAT_INTERFACE_SORTET[diFor2].proIsError < ayAT_INTERFACE_SORTET[diFor2 + 1].proIsError THEN
                    ITF_AT_Temp                         := ayAT_INTERFACE_SORTET[diFor2];
                    ayAT_INTERFACE_SORTET[diFor2]       := ayAT_INTERFACE_SORTET[diFor2 + 1];
                    ayAT_INTERFACE_SORTET[diFor2 + 1]   := ITF_AT_Temp;    
                ELSIF NOT ayAT_INTERFACE_SORTET[diFor2].proIsError THEN
                    IF ayAT_INTERFACE_SORTET[diFor2].proIsWarning < ayAT_INTERFACE_SORTET[diFor2 + 1].proIsWarning THEN
                        ITF_AT_Temp                         := ayAT_INTERFACE_SORTET[diFor2];
                        ayAT_INTERFACE_SORTET[diFor2]       := ayAT_INTERFACE_SORTET[diFor2 + 1];
                        ayAT_INTERFACE_SORTET[diFor2 + 1]   := ITF_AT_Temp;    
                    ELSIF ayAT_INTERFACE_SORTET[diFor2].proIsEnabled < ayAT_INTERFACE_SORTET[diFor2 + 1].proIsEnabled THEN
                        ITF_AT_Temp                         := ayAT_INTERFACE_SORTET[diFor2];
                        ayAT_INTERFACE_SORTET[diFor2]       := ayAT_INTERFACE_SORTET[diFor2 + 1];
                        ayAT_INTERFACE_SORTET[diFor2 + 1]   := ITF_AT_Temp;     
                    END_IF;                                                       
                END_IF;
            END_IF;       
        END_FOR;      
    END_FOR;        
ELSE
    uiSort := 0;     
END_IF; 
IF uiSort = 0 AND stSearch = '' THEN
    xIsSortet := FALSE;  
ELSE
    xIsSortet := TRUE;  
END_IF
END_METHOD

METHOD metGetAntriebITF : ITF_SENSOR
VAR_INPUT
    iPos    :   INT;
END_VAR
IF TO_DINT(iPos) >= LOWER_BOUND(ayAT_INTERFACE,1) AND TO_DINT(iPos) <= UPPER_BOUND(ayAT_INTERFACE,1) THEN
    IF xIsSortet THEN
        metGetAntriebITF := ayAT_INTERFACE_SORTET[iPos];       
    ELSE
        metGetAntriebITF := ayAT_INTERFACE[iPos];       
	END_IF   
END_IF
END_METHOD

END_FUNCTION_BLOCK

// 21 Interface/ITF_SENSOR_COLLECTOR
INTERFACE ITF_SENSOR_COLLECTOR

PROPERTY proBufferError : BOOL
GET
END_GET
END_PROPERTY

METHOD metGetAntriebITF : ITF_SENSOR
VAR_INPUT
    iPos    :   INT;
END_VAR
END_METHOD

PROPERTY proMissedBuffer : DINT
GET
END_GET
END_PROPERTY

PROPERTY proMin : INT
GET
END_GET
END_PROPERTY

PROPERTY proMax : UINT
GET
END_GET
END_PROPERTY

PROPERTY proaySensorTabelle : ARRAY[1..Parameter.iMaxSensor] OF ITF_SENSOR_TABELLE_INFO
GET
END_GET
END_PROPERTY

METHOD metSortArray
VAR_INPUT
    stSearch    :   STRING;
    uiSort      :   UINT;
END_VAR
END_METHOD

END_INTERFACE

// 30 Program Organization Units/fc's/fcGetBigerStringValue
FUNCTION fcGetBigerStringValue : INT
VAR_INPUT
    st1     :   STRING(255);
    st2     :   STRING(255);
END_VAR
VAR
    diFor: DINT;
    diMax: DINT;
END_VAR

IF LEN(st1) > LEN(st2) THEN
    diMax := LEN(st2); 
    fcGetBigerStringValue := 1;
ELSIF LEN(st1) < LEN(st2) THEN
    diMax := LEN(st1);
    fcGetBigerStringValue := 2;     
ELSE
    diMax := LEN(st1);    
END_IF;
FOR diFor := 0 TO  diMax DO
    IF st1[diFor] > st2[diFor] THEN
        fcGetBigerStringValue := 1;  
        EXIT; 
    ELSIF st1[diFor] < st2[diFor] THEN
        fcGetBigerStringValue := 2;  
        EXIT;
    END_IF;
END_FOR;

END_FUNCTION

// 30 Program Organization Units/fc's/AlarmControll/fcLowControl
FUNCTION fcLowControl : BOOL
VAR_INPUT
    xEn         :   BOOL;
    rIst        :   REAL;
    rLow        :   REAL;
    rHyst       :   REAL;
    xTrig       :   BOOL;       
END_VAR
VAR_OUTPUT
END_VAR
VAR
END_VAR

IF xTrig AND xEn THEN
   fcLowControl := rIst <= rLow + rHyst;
ELSIF xEn THEN
   fcLowControl := rIst <= rLow;
ELSE 
   fcLowControl := FALSE;
END_IF;

END_FUNCTION

// 30 Program Organization Units/fc's/AlarmControll/fcHighControl
FUNCTION fcHighControl : BOOL
VAR_INPUT
    xEn         :   BOOL;
    rIst        :   REAL;
    rHigh       :   REAL;
    rHyst       :   REAL;
    xTrig       :   BOOL;
END_VAR

IF xTrig AND xEn THEN
   fcHighControl := rIst >= rHigh - rHyst;
ELSIF xEn THEN
   fcHighControl := rIst >= rHigh;
ELSE
   fcHighControl := FALSE;
END_IF;

END_FUNCTION

// 30 Program Organization Units/fc's/Visu/fcCheckQuerryAndIconReturn
FUNCTION fcCheckQuerryAndIconReturn : BOOL
VAR_INPUT
	_ITF_IN			: 	ITF_SENSOR;
	_uiIconNr_IN	:	UINT;
END_VAR

IF __QUERYINTERFACE(_ITF_IN,_ITF_IN) THEN
	fcCheckQuerryAndIconReturn := TRUE;	
	_ITF_IN.proAtIconNr := _uiIconNr_IN;
ELSE
	fcCheckQuerryAndIconReturn :=  FALSE;
END_IF

END_FUNCTION

// 40 Visualizations/COLLECTOR/VIS_SENSOR_COLLECTOR
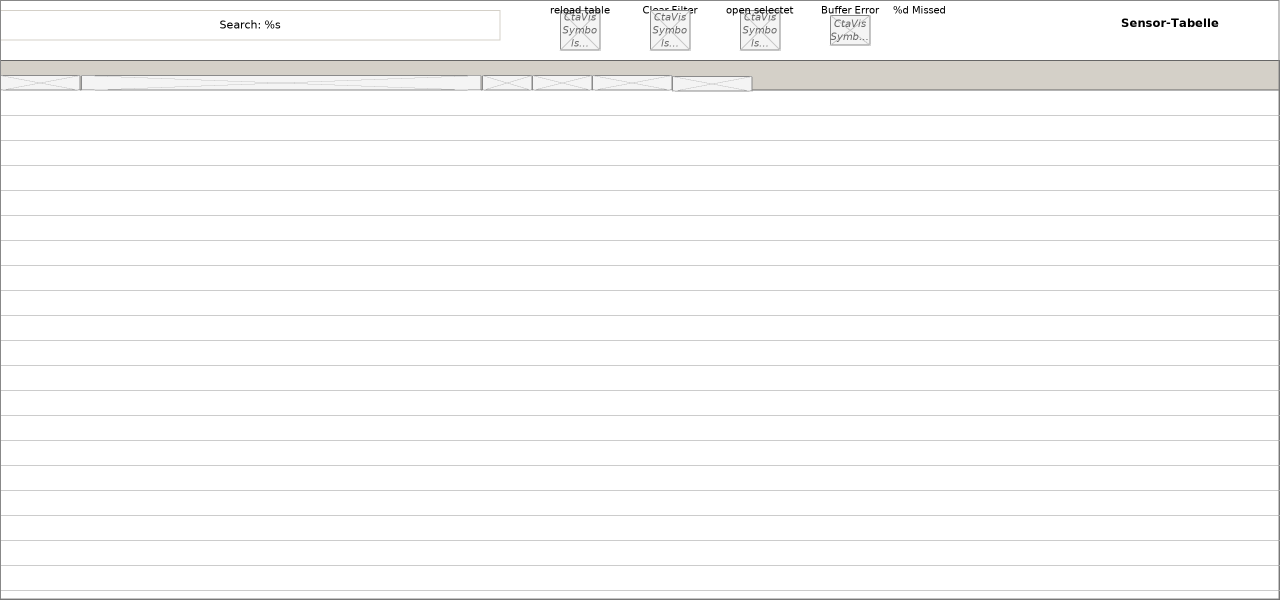
VISUALIZATION VIS_SENSOR_COLLECTOR  // 1280x600
    Frame (0,0 1280x600), invisible if: NOT GVL_SENSOR.xValidData
        shows VIS_SENSOR_COLLECTOR_TEMP(aySensorTabellenInfo := GVL_SENSOR.fbSENSOR_COLLECTOR.proaySensorTabelle, uiMax := GVL_SENSOR.fbSensor_Collector.proMax, ITF_SENSOR_COLLECTOR := GVL_SENSOR.fbSENSOR_COLLECTOR)
END_VISUALIZATION

// 40 Visualizations/COLLECTOR/Help Funktionen/SelSort
VISUALIZATION SelSort  // 15x30
VAR_IN_OUT
	uiSel                       :   UINT;
END_VAR
VAR_INPUT
    stSearch                    :   STRING;    
    ITF_SENSOR_COLLECTOR       : ITF_SENSOR_COLLECTOR;
END_VAR
VAR_INPUT CONSTANT
    uiValue             :   UINT;
END_VAR
    Frame (0,15 15x15), invisible if: uiValue <> uiSel
        shows SortPfeil()
    Rectangle (0,0 15x30)
        OnMouseClick: execute {
            IF uiSel <> uiValue THEN
                uiSel   := uiValue;
            ELSE
                uiSel   := 0;
            END_IF
            ITF_SENSOR_COLLECTOR.metSortArray(stSearch,uiSel);
        }
END_VISUALIZATION

